# B&R Automation Studio project mappFramework (part 4)

#### FileMgr.st
```iecst
//***********************************************************************
// Copyright: B&R Industrial Automation GmbH
// Author: B&R Industrial Automation GmbH
// Created: April 12, 2022
// Description: Task for file management
//***********************************************************************

PROGRAM _INIT

	// Inititialize mapp function block
	MpFileManagerUIConnect.DeviceList.DeviceNames[0] := 'USER';
	MpFileManagerUIConnect.DeviceList.DeviceNames[1] := 'mappRecipeFiles';
	MpFileManagerUIConnect.DeviceList.DeviceNames[2] := 'mappAuditFiles';
	MpFileManagerUIConnect.DeviceList.DeviceNames[3] := 'mappReportFiles';
	MpFileManagerUIConnect.DeviceList.DeviceNames[4] := 'mappBackupFiles';
	MpFileManagerUIConnect.DeviceList.DeviceNames[5] := 'mappAlarmXFiles';
	MpFileManagerUIConnect.DeviceList.DeviceNames[6] := 'mappUserXFiles';
	MpFileManagerUISys.Enable := TRUE;
	MpFileManagerUISys.MpLink := ADR(gMpLinkFileManagerUIFile);
	MpFileManagerUISys.UIConnect := ADR(MpFileManagerUIConnect);
	MpFileManagerUISys.UISetup.FileListSize := SIZEOF(MpFileManagerUIConnect.File.List.Items) / SIZEOF(MpFileManagerUIConnect.File.List.Items[0]);
	MpFileManagerUISys();

	HmiFile.Status.DeleteStep := FILE_DISABLED;

	// Restored the retained values to the FIFO settings
	HmiFile.Parameters.Fifo := FifoSettingsRetain;
	// If the FIFO is disabled and parameters are 0, set default values
	IF NOT HmiFile.Parameters.Fifo.Enable THEN
		IF HmiFile.Parameters.Fifo.MaxFolderSize = 0 THEN
			HmiFile.Parameters.Fifo.MaxFolderSize := 1000;
		END_IF
		IF HmiFile.Parameters.Fifo.MaxNumberOfFiles = 0 THEN
			HmiFile.Parameters.Fifo.MaxNumberOfFiles := 20;
		END_IF
		IF HmiFile.Parameters.Fifo.ScanInterval = 0 THEN
			HmiFile.Parameters.Fifo.ScanInterval := 60;
		END_IF
		IF HmiFile.Parameters.Fifo.DeviceName = '' THEN
			HmiFile.Parameters.Fifo.DeviceName := 'USER';
		END_IF
	END_IF

	// Initialize which folders should exist
	PathCheck.DeviceList := MpFileManagerUIConnect.DeviceList;

	PathCheck.PrgName[0] := 'RecipeMgr';
	PathCheck.PrgName[1] := 'AuditMgr';
	PathCheck.PrgName[2] := 'ReportMgr';
	PathCheck.PrgName[3] := 'BackupMgr';
	PathCheck.PrgName[4] := 'AlarmMgr';
	PathCheck.PrgName[5] := 'UserXMgr';
	PathCheck.PrgName[6] := 'UsbMgr';
	PathCheck.PrgName[7] := 'UsbMgr';

	PathCheck.Folder[0] := 'Recipe';
	PathCheck.Folder[1] := 'Audit';
	PathCheck.Folder[2] := 'Report';
	PathCheck.Folder[3] := 'Backup';
	PathCheck.Folder[4] := 'AlarmX';
	PathCheck.Folder[5] := 'UserX';

	HmiFile.Status.DeviceDataProvider[0] := '{"value":"USER","text":"UserPath"}';
	HmiFile.Status.DeviceDataProvider[1] := '{"value":"mappRecipeFiles","text":"mappRecipeFiles"}';
	HmiFile.Status.DeviceDataProvider[2] := '{"value":"mappAuditFiles","text":"mappAuditFiles"}';
	HmiFile.Status.DeviceDataProvider[3] := '{"value":"mappReportFiles","text":"mappReportFiles"}';
	HmiFile.Status.DeviceDataProvider[4] := '{"value":"mappBackupFiles","text":"mappBackupFiles"}';
	HmiFile.Status.DeviceDataProvider[5] := '{"value":"mappAlarmXFiles","text":"mappAlarmXFiles"}';
	HmiFile.Status.DeviceDataProvider[6] := '{"value":"mappUserXFiles","text":"mappUserXFiles"}';

	// Calculate offset for potential additional USB devices
	FOR i := 0 TO ((SIZEOF(MpFileManagerUIConnect.DeviceList.DeviceNames) / SIZEOF(MpFileManagerUIConnect.DeviceList.DeviceNames[0])) - 1) DO
		IF MpFileManagerUIConnect.DeviceList.DeviceNames[i] <> '' THEN
			USBOffset := USBOffset + 1;
		END_IF
	END_FOR

END_PROGRAM

PROGRAM _CYCLIC

	// Call all cyclic actions
	FormatDeviceDataProvider;
	FileManager;
	FIFOOperation;

	// Error reset
	IF NOT MpFileManagerUISys.Error THEN
		MpFileManagerUISys.ErrorReset := FALSE;
	END_IF

	// Assign MpLinks and address references
	MpFileManagerUISys.MpLink := ADR(gMpLinkFileManagerUIFile);
	MpFileManagerUISys.UIConnect := ADR(MpFileManagerUIConnect);
	MpFileManagerUI_FIFO.MpLink := ADR(gMpLinkFileManagerUIFile_FIFO);

	// Call function blocks
	MpFileManagerUISys();
	MpFileManagerUI_FIFO();

END_PROGRAM

PROGRAM _EXIT

	// Disable the function blocks to unlink the MpLink
	MpFileManagerUISys.Enable := FALSE;
	MpFileManagerUI_FIFO.Enable := FALSE;

	// Call function blocks
	MpFileManagerUISys();
	MpFileManagerUI_FIFO();

END_PROGRAM
```

#### HMIActions.st
```iecst
ACTION FormatDeviceDataProvider:

	// Select CF device if USB device is not available
	FOR i := 0 TO IDX_USB_DEV_LIST DO
		tempIdx := (i + USBOffset);

		IF gUSBAvailable[i] THEN

			HmiFile.Status.DeviceDataProvider[tempIdx] := '{"value":"USB';
			brsitoa(i + 1, ADR(HmiFile.Status.DeviceDataProvider[tempIdx]) + brsstrlen(ADR(HmiFile.Status.DeviceDataProvider[tempIdx])));

			brsstrcat(ADR(HmiFile.Status.DeviceDataProvider[tempIdx]), ADR('","text":"USB'));
			brsitoa(i + 1, ADR(HmiFile.Status.DeviceDataProvider[tempIdx]) + brsstrlen(ADR(HmiFile.Status.DeviceDataProvider[tempIdx])));
			brsstrcat(ADR(HmiFile.Status.DeviceDataProvider[tempIdx]), ADR('"}'));

			PathCheck.DeviceList.DeviceNames[tempIdx] := 'USB';
			brsitoa(i + 1, ADR(PathCheck.DeviceList.DeviceNames[tempIdx]) + brsstrlen(ADR(PathCheck.DeviceList.DeviceNames[tempIdx])));
		ELSE
			brsmemset(ADR(HmiFile.Status.DeviceDataProvider[tempIdx]), 0, SIZEOF(HmiFile.Status.DeviceDataProvider[tempIdx]));
			brsmemset(ADR(PathCheck.DeviceList.DeviceNames[tempIdx]), 0, SIZEOF(PathCheck.DeviceList.DeviceNames[tempIdx]));
		END_IF
	END_FOR

	//Check initilized folder for existance and remove any from the device list that don't exist
	MaxDeviceNameIndex := ((SIZEOF(MpFileManagerUIConnect.DeviceList.DeviceNames) / SIZEOF(MpFileManagerUIConnect.DeviceList.DeviceNames[0])) - 1);
	NextOpenIndex := 0;
	FOR index := 0 TO MaxDeviceNameIndex DO
		IdentStatus := ST_ident(ADR(PathCheck.PrgName[index]),0,ADR(Ident));
		//Assign device name to next available slot in table according to if the path is valid
		IF (IdentStatus = 0) THEN		//path is valid
			MpFileManagerUIConnect.DeviceList.DeviceNames[NextOpenIndex] := PathCheck.DeviceList.DeviceNames[index + 1];
			NextOpenIndex := NextOpenIndex + 1;
		END_IF;
		//Clear the remaining index slots with invalid path checks
		IF index > NextOpenIndex THEN
			MpFileManagerUIConnect.DeviceList.DeviceNames[index] := '';
		END_IF
	END_FOR;

	// Configure visible device list
	HmiFile.Status.TableConfig[0] := '{ "specRows": [{"from":';
	FOR i := 0 TO MaxDeviceNameIndex DO
		IF MpFileManagerUIConnect.DeviceList.DeviceNames[i] <> '' THEN
			DeviceCount := i + 1;
		END_IF
	END_FOR
	brsitoa((DeviceCount), ADR(HmiFile.Status.TableConfig[0]) + brsstrlen(ADR(HmiFile.Status.TableConfig[0])));
	brsstrcat(ADR(HmiFile.Status.TableConfig[0]), ADR(',"to":9, "visible":false}]}'));

	// Configure visible file list
	HmiFile.Status.TableConfig[1] := '{ "specRows": [{"from":';
	brsitoa((MpFileManagerUIConnect.File.PathInfo.FileCount + MpFileManagerUIConnect.File.PathInfo.FolderCount), ADR(HmiFile.Status.TableConfig[1]) + brsstrlen(ADR(HmiFile.Status.TableConfig[1])));
	brsstrcat(ADR(HmiFile.Status.TableConfig[1]), ADR(',"to":49, "visible":false}]}'));

	// Create device data provider for FIFO drop down
	FOR i := 0 TO MaxDeviceNameIndex DO
		IF (MpFileManagerUIConnect.DeviceList.DeviceNames[i] <> '') THEN
			HmiFile.Status.DeviceDataProvider[i] := '{"value":"';
			brsstrcat(ADR(HmiFile.Status.DeviceDataProvider[i]), ADR(MpFileManagerUIConnect.DeviceList.DeviceNames[i]));
			brsstrcat(ADR(HmiFile.Status.DeviceDataProvider[i]), ADR('","text":"'));
			brsstrcat(ADR(HmiFile.Status.DeviceDataProvider[i]), ADR(MpFileManagerUIConnect.DeviceList.DeviceNames[i]));
			brsstrcat(ADR(HmiFile.Status.DeviceDataProvider[i]), ADR('"}'));
		ELSE
			brsmemset(ADR(HmiFile.Status.DeviceDataProvider[i]), 0, SIZEOF(HmiFile.Status.DeviceDataProvider[i]));
		END_IF
	END_FOR

END_ACTION

ACTION FileManager:

	MpFileManagerUI_0.MpLink := ADR(gMpLinkFileManagerUIFile);
	MpFileManagerUI_0.UIConnect := ADR(MpFileManagerUIConnect);
	MpFileManagerUI_0();

	FOR i := 0 TO ((SIZEOF(HmiFile.Status.FileNames)/SIZEOF(HmiFile.Status.FileNames[0])) - 1) DO
		HmiFile.Status.FileNames[i] := MpFileManagerUIConnect.File.List.Items[i].Name;
		HmiFile.Status.TimeStamps[i] := MpFileManagerUIConnect.File.List.Items[i].LastModified;
		HmiFile.Status.Size[i] := REAL_TO_UDINT(UDINT_TO_REAL(MpFileManagerUIConnect.File.List.Items[i].Size) * 0.001);

		// Set image array based on item type
		IF MpFileManagerUIConnect.File.List.Items[i].IsFolder THEN
			HmiFile.Status.Type[i] := FOLDER;
		ELSIF NOT MpFileManagerUIConnect.File.List.Items[i].IsFolder AND MpFileManagerUIConnect.File.List.Items[i].IsSelected THEN
			HmiFile.Status.Type[i] := FILE_SELECTED;
		ELSE
			HmiFile.Status.Type[i] := FILE;
		END_IF

		// Set file selected when the table is clicked Single and MultiSelect
		IF (MpFileManagerUIConnect.File.MultiSelect = FALSE) THEN
			MpFileManagerUIConnect.File.List.Items[i].IsSelected := (i = HmiFile.Status.SelectedIndex);
		ELSIF (MpFileManagerUIConnect.File.MultiSelect = TRUE) AND (HmiFile.Commands.MultiSelect = TRUE) THEN
			IF (i = HmiFile.Status.SelectedIndex) AND NOT MpFileManagerUIConnect.File.List.Items[i].IsSelected THEN
				MpFileManagerUIConnect.File.List.Items[i].IsSelected := TRUE;
				HmiFile.Commands.MultiSelect := FALSE;
			ELSIF (i = HmiFile.Status.SelectedIndex) AND MpFileManagerUIConnect.File.List.Items[i].IsSelected THEN
				MpFileManagerUIConnect.File.List.Items[i].IsSelected := FALSE;
				HmiFile.Commands.MultiSelect := FALSE;
			END_IF
		END_IF
	END_FOR

	// Read currently selected device name for HMI
	IF (MpFileManagerUIConnect.DeviceList.SelectedIndex >= (SIZEOF(MpFileManagerUIConnect.DeviceList.DeviceNames) / SIZEOF(MpFileManagerUIConnect.DeviceList.DeviceNames[0]))) THEN
		MpFileManagerUIConnect.DeviceList.SelectedIndex := 0;
	END_IF
	HmiFile.Status.DeviceName := MpFileManagerUIConnect.DeviceList.DeviceNames[MpFileManagerUIConnect.DeviceList.SelectedIndex];

	// Read if current selected object is folder
	IF (HmiFile.Status.SelectedIndex >= (SIZEOF(MpFileManagerUIConnect.File.List.Items) / SIZEOF(MpFileManagerUIConnect.File.List.Items[0]))) THEN
		HmiFile.Status.SelectedIndex := 0;
	END_IF
	HmiFile.Status.IsFolder := MpFileManagerUIConnect.File.List.Items[HmiFile.Status.SelectedIndex].IsFolder;

	// Control the folder structure when entering and leaving folders
	IF (HmiFile.Commands.EnterFolder) AND MpFileManagerUIConnect.File.List.Items[HmiFile.Status.SelectedIndex].IsFolder THEN
		HmiFile.Commands.EnterFolder := FALSE;
		MpFileManagerUIConnect.File.EnterFolder := TRUE;
		FolderDepthCount := FolderDepthCount + 1;
	ELSE
		HmiFile.Commands.EnterFolder := FALSE;
	END_IF

	IF EDGEPOS(HmiFile.Commands.FolderUp) AND (HmiFile.Status.BackButton > 0) THEN
		HmiFile.Commands.FolderUp := FALSE;
		MpFileManagerUIConnect.File.FolderUp := TRUE;
		FolderDepthCount := FolderDepthCount - 1;
	END_IF

	HmiFile.Status.BackButton := (FolderDepthCount > 0);
	HmiFile.Status.DefaultFileSelected := ((MpFileManagerUIConnect.File.List.Items[HmiFile.Status.SelectedIndex].Name = CONCAT(DEFAULT_PARAMETERS,PARAMETERS_FILE_EXTENSION)) OR
																				(MpFileManagerUIConnect.File.List.Items[HmiFile.Status.SelectedIndex].Name = CONCAT(DEFAULT_MACHINE_CONFIGURATION,
																				MACHINE_CONFIG_FILE_EXTENSION))) AND MpFileManagerUIConnect.DeviceList.SelectedIndex = 0;

END_ACTION
```

### Package Logical/Infrastructure/Usb - Package for USB handling for mapp Framework

### Program Logical/Infrastructure/Usb/UsbMgr (IEC)

#### UsbMgr.st - Cyclic code
```iecst
//*********************************************************************************
// Copyright: B&R Industrial Automation GmbH
// Author: B&R Industrial Automation GmbH
// Created: April 12, 2022
// Description: This task automatically detects and (un)links USB storage devices
//*********************************************************************************

PROGRAM _INIT
END_PROGRAM

PROGRAM _CYCLIC

	CASE StateMachine OF
		// -----------------------------------------------------------------------------------------------------------
		// Wait state
		// -----------------------------------------------------------------------------------------------------------
		USB_WAIT:
			// Refresh USB data every X seconds when enabled
			Node := 1;
			USB.Status := ERR_OK;
			IF USB.Cmd.AutoScan THEN
				RefreshTimer(IN := 1, PT := USB.Par.RefreshInterval);
				// Get new USB data
				IF(RefreshTimer.Q) THEN
					RefreshTimer(IN := 0);
					USB.Status := ERR_FUB_BUSY;
					brsmemset(ADR(UsbData), 0, SIZEOF(UsbData));
					StateMachine := USB_CREATE_NODE_ID_LIST;
				END_IF
			ELSE
				RefreshTimer(IN := 0);
			END_IF
			// Refresh USB data every X seconds when enabled
			IF USB.Cmd.ErrorReset THEN
				StateMachine := USB_ERROR;
			END_IF

			FOR i := 0 TO IDX_USB_DEV_LIST DO
				gUSBAvailable[i] := USB.Par.IsConnected[i+1];
			END_FOR

			// -----------------------------------------------------------------------------------------------------------
			// Get USB device list
			// -----------------------------------------------------------------------------------------------------------
		USB_CREATE_NODE_ID_LIST:
			GetUsbNodeList.enable := 1;
			GetUsbNodeList.pBuffer := ADR(NodeIdBuffer);
			GetUsbNodeList.bufferSize := SIZEOF(NodeIdBuffer);
			GetUsbNodeList.filterInterfaceClass := asusb_CLASS_MASS_STORAGE;
			GetUsbNodeList.filterInterfaceSubClass := 0;
			GetUsbNodeList;

			// --------------------------------------------------------------------------------------------------------------------
			// Success
			IF GetUsbNodeList.status = 0 THEN
				StateMachine := USB_READ_DEVICE_DATA;
				Node := 1;
				// No USB devices found
			ELSIF GetUsbNodeList.status = asusbERR_USB_NOTFOUND THEN
				// Unlink old device if it is gone now otherwise wait for next round
				FOR i:=1 TO MAX_IDX_USB_DEV_LIST DO
					IF(USB.Par.IsConnected[i]) THEN
						Node := 1;
						StateMachine := USB_CHECK_LINKED;
						RETURN;
					END_IF
				END_FOR;
				StateMachine := USB_WAIT;
				// Error
			ELSIF GetUsbNodeList.status <> ERR_FUB_BUSY THEN
				USB.Status := GetUsbNodeList.status;
				USB.Err.State := StateMachine;
				IF GetUsbNodeList.status = asusbERR_BUFSIZE THEN
					USB.Err.Text := 'maximum number of devices reached';
				ELSE
					USB.Err.Text := 'error getting device list';
				END_IF;
				StateMachine := USB_ERROR;
			END_IF;
			// -----------------------------------------------------------------------------------------------------------
			// Get device information
			// -----------------------------------------------------------------------------------------------------------
		USB_READ_DEVICE_DATA:
			GetUsbNode.enable := 1;
			GetUsbNode.nodeId := NodeIdBuffer[Node];
			GetUsbNode.pBuffer := ADR(UsbData[Node]);
			GetUsbNode.bufferSize := SIZEOF (UsbData[Node]);
			GetUsbNode;

			// --------------------------------------------------------------------------------------------------------------------
			// Success
			IF GetUsbNode.status = 0 THEN
				// Make sure we have enough space to store USB data, proceed with next StateMachine when all devices are detetced
				IF (Node = GetUsbNodeList.listNodes) OR (Node = MAX_IDX_USB_DEV_LIST) THEN
					Node := 1;
					StateMachine := USB_CHECK_LINKED;
					// Get next USB device
				ELSE
					Node := Node + 1;
				END_IF;
				// Error
			ELSIF GetUsbNode.status <> ERR_FUB_BUSY THEN
				USB.Status := GetUsbNode.status;
				USB.Err.State := StateMachine;
				USB.Err.Text := 'error getting device data';
				StateMachine := USB_ERROR;
			END_IF;
			// -----------------------------------------------------------------------------------------------------------
			// Check if linked device are still present
			// -----------------------------------------------------------------------------------------------------------
		USB_CHECK_LINKED:
			// Proceed to new devices when last device was checked
			IF(Node > MAX_IDX_USB_DEV_LIST) THEN
				Node := 1;
				StateMachine := USB_LINK_NEW;
				RETURN;
			END_IF

			// -----------------------------------------------------------------------------------------------------------
			// Check if device is still active
			IsLinked := FALSE;
			FOR i:=1 TO MAX_IDX_USB_DEV_LIST DO
				// Compare old and new data
				IF(brsmemcmp(ADR(UsbDataOld[Node]), ADR(UsbData[i]), SIZEOF(UsbData[i])) = 0) AND
					(NOT USB.Par.IgnoreDongle OR (USB.Par.IgnoreDongle AND UsbData[i].productId <> BrProductId AND UsbData[i].vendorId <> BrVendorId)) THEN
					// Clear data, mark as linked and EXIT loop
					brsmemset(ADR(UsbData[i]), 0, SIZEOF(UsbData[i]));
					IsLinked := TRUE;
					EXIT;
				END_IF
			END_FOR;

			// -----------------------------------------------------------------------------------------------------------
			// Find next linked device
			IF(IsLinked OR UsbDataOld[Node].interfaceClass = 0) THEN
				IF(Node < MAX_IDX_USB_DEV_LIST) THEN
					Node := Node + 1;
					WHILE(Node < MAX_IDX_USB_DEV_LIST AND UsbDataOld[Node].interfaceClass = 0) DO
						Node := Node + 1;
					END_WHILE;
					IF(Node = MAX_IDX_USB_DEV_LIST AND UsbDataOld[Node].interfaceClass = 0) THEN
						Node := Node + 1;
					END_IF
				ELSE
					Node := Node + 1;
				END_IF
				// Unlink device if it is missing
			ELSE
				StateMachine := USB_UNLINK_DEVICE;
			END_IF
			// -----------------------------------------------------------------------------------------------------------
			// Link new devices
			// -----------------------------------------------------------------------------------------------------------
		USB_LINK_NEW:
			// Return to wait state when last device was checked
			IF(Node > MAX_IDX_USB_DEV_LIST) THEN
				StateMachine := USB_WAIT;
				RETURN;
			END_IF

			// -----------------------------------------------------------------------------------------------------------
			// Find next new device
			IF(UsbData[Node].interfaceClass <> 0) THEN
				IF(USB.Par.IgnoreDongle OR (UsbData[Node].productId <> BrProductId AND UsbData[Node].vendorId <> BrVendorId)) THEN
					StateMachine := USB_LINK_DEVICE;
					RETURN;
				END_IF
			END_IF
			Node := Node + 1;
			// -----------------------------------------------------------------------------------------------------------
			// Link device
			// -----------------------------------------------------------------------------------------------------------
		USB_LINK_DEVICE:
			// Find empty slot
			FOR i:=1 TO MAX_IDX_USB_DEV_LIST DO
				IF(UsbDataOld[i].interfaceClass = 0) THEN
					EXIT;
				END_IF
			END_FOR;
			// No more slot available
			IF(i = MAX_IDX_USB_DEV_LIST AND UsbDataOld[i].interfaceClass <> 0) THEN
				USB.Status := ERR_MAX_DEVICE;
				USB.Err.State := StateMachine;
				USB.Err.Text := 'maximum number of device reached';
				StateMachine := USB_ERROR;
				RETURN;
			END_IF
			// Create device string
			brsstrcpy(ADR(DevicePara), ADR('/DEVICE='));
			brsstrcat(ADR(DevicePara), ADR(UsbData[Node].ifName));
			brsstrcpy(ADR(DeviceName), ADR('USB'));
			brsitoa(i, ADR(tmpSTR));
			brsstrcat(ADR(DeviceName), ADR(tmpSTR));
			// Link device
			DevLinkSys.enable := 1;
			DevLinkSys.pDevice := ADR(DeviceName);
			DevLinkSys.pParam := ADR(DevicePara);
			DevLinkSys;

			// --------------------------------------------------------------------------------------------------------------------
			// Success
			IF DevLinkSys.status = 0 THEN
				// Store data for new device
				brsmemcpy(ADR(UsbDataOld[i]), ADR(UsbData[Node]), SIZEOF(UsbData[Node]));
				USB.Par.IsConnected[i] := TRUE;
				LinkHandle[i] := DevLinkSys.handle;
				Node := Node + 1;
				StateMachine := USB_LINK_NEW;
				// Error
			ELSIF DevLinkSys.status <> ERR_FUB_BUSY THEN
				USB.Status := DevLinkSys.status;
				USB.Err.State := StateMachine;
				USB.Err.Text := 'error linking device';
				StateMachine := USB_ERROR;
			END_IF;
			// -----------------------------------------------------------------------------------------------------------
			// UnLink device
			// -----------------------------------------------------------------------------------------------------------
		USB_UNLINK_DEVICE:
			DevUnlinkSys.enable := 1;
			DevUnlinkSys.handle := LinkHandle[Node];
			DevUnlinkSys;

			// --------------------------------------------------------------------------------------------------------------------
			// Success
			IF DevUnlinkSys.status = 0 THEN
				// Clear data
				brsmemset(ADR(UsbDataOld[Node]), 0, SIZEOF(UsbDataOld[Node]));
				USB.Par.IsConnected[Node] := FALSE;
				LinkHandle[Node] := 0;
				// Find next linked device
				WHILE(Node < MAX_IDX_USB_DEV_LIST AND UsbDataOld[Node].interfaceClass = 0) DO
					Node := Node + 1;
				END_WHILE;
				IF(Node = MAX_IDX_USB_DEV_LIST AND UsbDataOld[Node].interfaceClass = 0) THEN
					Node := Node + 1;
				END_IF
				StateMachine := USB_CHECK_LINKED;
				// Error
			ELSIF DevUnlinkSys.status <> ERR_FUB_BUSY THEN
				// Clear data
				brsmemset(ADR(UsbDataOld[Node]), 0, SIZEOF(UsbDataOld[Node]));
				USB.Par.IsConnected[Node] := FALSE;
				LinkHandle[Node] := 0;

				brsitoa(Node, ADR(tmpSTR));
				USB.Status := DevUnlinkSys.status;
				USB.Err.State := StateMachine;
				USB.Err.Text := 'error unlinking device no ';
				brsstrcat(ADR(USB.Err.Text), ADR(tmpSTR));
				StateMachine := USB_ERROR;
			END_IF;
			// -----------------------------------------------------------------------------------------------------------
			// Error state
			// -----------------------------------------------------------------------------------------------------------
		USB_ERROR:
			// Get more error information
			IF(USB.Status = 0) THEN
				USB.Status := FileIoGetSysError();
			END_IF

			// Unlink device
			IF(USB.Err.State = USB_LINK_DEVICE) THEN
				DevUnlinkSys.enable := 1;
				DevUnlinkSys.handle := DevLinkSys.handle;
				DevUnlinkSys;
			END_IF

			// Reset error
			IF(USB.Cmd.ErrorReset AND DevUnlinkSys.status <> ERR_FUB_BUSY) THEN
				USB.Cmd.ErrorReset := FALSE;
				brsmemset(ADR(USB.Err), 0, SIZEOF(USB.Err));
				StateMachine := USB_WAIT;
			END_IF
	END_CASE;

END_PROGRAM

PROGRAM _EXIT
	FOR i:=1 TO MAX_IDX_USB_DEV_LIST DO
		REPEAT
			DevUnlinkSys.enable := 1;
			DevUnlinkSys.handle := LinkHandle[i];
			DevUnlinkSys;
			UNTIL DevUnlinkSys.status <> ERR_FUB_BUSY
		END_REPEAT;
	END_FOR;
END_PROGRAM
```

#### UsbMgr.typ
```iecst
TYPE
	UsbStateEnum :
		(
		USB_WAIT, (*Wait for starting the Function chain*)
		USB_CREATE_NODE_ID_LIST, (*Create a list of Node-IDs from all active USB devices*)
		USB_READ_DEVICE_DATA, (*Read out the specific data from the Node-IDs*)
		USB_CHECK_LINKED, (*Check if device is still connected*)
		USB_LINK_NEW,
		USB_LINK_DEVICE, (*Link file device*)
		USB_UNLINK_DEVICE, (*Unlink the File Device from specific path*)
		USB_ERROR (*Jump to this step in every case of Error occuring in the Function chain*)
		);
	UsbCmdType : 	STRUCT
		AutoScan : BOOL := TRUE; (*Scan USB ports automatically*)
		ErrorReset : BOOL; (*Reset error*)
	END_STRUCT;
	UsbParType : 	STRUCT
		IgnoreDongle : BOOL := TRUE; (*Ignoe B&R license dongle*)
		RefreshInterval : UINT := 300; (*Intervall timer for USB device refresh*)
		IsConnected : ARRAY[0..MAX_IDX_USB_DEV_LIST]OF BOOL; (*Shows if a USB stick is connected*)
	END_STRUCT;
	UsbErrType : 	STRUCT
		State : UsbStateEnum; (*State where the error occured*)
		Text : STRING[80]; (*Error text*)
	END_STRUCT;
	UsbMainType : 	STRUCT
		Cmd : UsbCmdType; (*Command structure*)
		Par : UsbParType; (*Parameter structure*)
		Err : UsbErrType; (*Error structure*)
		Status : UINT; (*Current status*)
	END_STRUCT;
END_TYPE
```

#### UsbMgr.var - Data for read_data Task
```iecst
(*Function Blocks*)
VAR
	RefreshTimer : TON;
	GetUsbNodeList : UsbNodeListGet; (*Type of FUB UsbNodeListGet*)
	GetUsbNode : UsbNodeGet; (*Type of FUB UsbNodeGet*)
	DevLinkSys : DevLink; (*Type of FUB DevLink*)
	DevUnlinkSys : DevUnlink; (*Type of FUB DevUnlink*)
END_VAR
(*Constants*)
VAR CONSTANT
	BrVendorId : UINT := 1615; (*B&R vendor id*)
	BrProductId : UINT := 1001; (*B&R dongle product id*)
	ERR_MAX_DEVICE : UINT := 50000; (*Maximum number of dongles reached*)
END_VAR
(*Structure Types*)
VAR
	USB : UsbMainType;
	StateMachine : UsbStateEnum; (*State machine*)
	UsbData : ARRAY[1..MAX_IDX_USB_DEV_LIST] OF usbNode_typ; (*Data of all available USB devices*)
	UsbDataOld : ARRAY[1..MAX_IDX_USB_DEV_LIST] OF usbNode_typ; (*Old data of all available USB devices*)
END_VAR
(*Variables*)
VAR
	DevicePara : STRING[80]; (*Connection path of USB device*)
	DeviceName : STRING[40]; (*Connection path of USB device*)
	LinkHandle : ARRAY[1..MAX_IDX_USB_DEV_LIST] OF UDINT; (*Link handle for USB device*)
	NodeIdBuffer : ARRAY[1..MAX_IDX_USB_DEV_LIST] OF UDINT; (*Different nodeIDs saved in array-elements*)
	IsLinked : BOOL; (*Helper variable that indicates that a USB stick is linked*)
	Node : USINT; (*Node number*)
	i : USINT;
	tmpSTR : STRING[10];
END_VAR
```

### Package Logical/Infrastructure/Recipe - Package for mapp Recipe Framework

### Program Logical/Infrastructure/Recipe/RecipeMgr (IEC) - Recipe manager

#### RecipeMgr.typ
```iecst
(*Structure types*)

TYPE
	RecipeHmiInterfaceType : 	STRUCT  (*Structure to hold commands, parameters and status from the HMI*)
		Commands : RecipeCommandsType; (*Structure to hold the commands from the HMI*)
		Parameters : RecipeParametersType; (*Structure to hold the parameters for the HMI*)
		Status : RecipeStatusType; (*Structure to hold status information from the mapp View HMI*)
	END_STRUCT;
	RecipeCommandsType : 	STRUCT  (*Structure to hold the commands from the HMI*)
		LoadRecipe : BOOL; (*Load recipe*)
		SaveSelectedRecipe : BOOL; (*Save the selected recipe (which is not necessarily the active recipe)*)
		CreateRecipe : BOOL; (*Create recipe*)
		ResetPreview : BOOL; (*Reset the preview to empty/zeros in the event of an invalid recipe*)
	END_STRUCT;
	RecipeParametersType : 	STRUCT  (*Structure to hold the parameters for the HMI*)
		Category : STRING[30]; (*Current category*)
		DeviceName : STRING[50]; (*Selected file device name*)
		FileName : STRING[255]; (*Recipe file name*)
	END_STRUCT;
	RecipeStatusType : 	STRUCT  (*Structure to hold status information from the mapp View HMI*)
		PreviewCase : PreviewCaseEnum; (*State machine step for loading previews*)
		HMIcommand : RecipeHmiStepEnum; (*State machine step for HMI commands*)
		LastLoadedConfigRecipe : STRING[255]; (*Last loaded configuration recipe*)
		LastLoadedProductRecipe : STRING[255]; (*Last loaded product recipe*)
		ProductRecipeLoaded : BOOL; (*Product recipe was loaded*)
		ConfigRecipeLoaded : BOOL; (*Config recipe was loaded*)
		PreviousRangeStart : REAL; (*Scroll range temp variables*)
		PreviousRangeEnd : REAL; (*Scroll range temp variables*)
		LastMaxSelection : UINT; (*The previous maximum number of recipes*)
		SelectedIndex : UINT; (*The currently selected index*)
		LastSelectedIndex : UINT; (*The previous selected index*)
		LastStatus : MpRecipeUIStatusEnum; (*The previous UI status*)
		EditDialogOpened : BOOL; (*Flag that the edit dialog box was opened*)
		CreateDialogOpened : BOOL; (*Flag that the create dialog box was opened*)
		DefaultConfig : STRING[255]; (*Name of the default configuration*)
		DefaultRecipe : STRING[255]; (*Name of the default recipe*)
		FileDuplicate : BOOL; (*Recipe file already exists, warn the user.*)
		FilesAvailable : BOOL; (*Control access to widget when no files are available*)
		InvalidRecipe : BOOL; (*The selected recipe cannot be previewed*)
		LoadingRecipeList : BOOL; (*The recipe list is loading*)
		MachineSettingsRecipeMissing : BOOL; (*Flag for if the default machine settings recipe is not present*)
		ParameterRecipeMissing : BOOL; (*Flag for if the default parameters recipe is not present*)
		DeviceValid : BOOL; (*Flag for whether FileDevice is valid. Prevents user from being prompted to load default recipe.*)
		LoadAllowed : BOOL; (*Flag for whether you can load a recipe. Recipe must exist and be valid. *)
		DeviceDataProvider : ARRAY[0..MAX_IDX_FILE_DEV]OF STRING[100]; (*File device data provider*)
		TableConfig : STRING[120]; (*Table configuration *)
		SelectedRecipe : STRING[255]; (*The name of the selected recipe*)
		DefaultRecipeSelected : BOOL; (*The default recipe is selected*)
		RecipeContentLoaded : BOOL; (*Recipe content is loading and previous selection is restored*)
	END_STRUCT;
	RecipeRetainType : 	STRUCT  (*Structure to hold parameters for retain after restart *)
		LastLoadedConfigRecipe : STRING[255]; (*Last loaded configuration recipe*)
		LastLoadedProductRecipe : STRING[255]; (*Last loaded product recipe*)
	END_STRUCT;
	ParametersType : 	STRUCT  (*Demo / starter structure for machine parameters*)
		AddParametersHere1 : BOOL; (*Add your parameteres here *)
		AddParametersHere2 : STRING[80]; (*Add your parameteres here *)
		AddParametersHere3 : REAL; (*Add your parameteres here *)
		AddParametersHere4 : REAL; (*Add your parameteres here *)
		AddParametersHere5 : REAL; (*Add your parameteres here *)
	END_STRUCT;
	MachineSettingsType : 	STRUCT  (*Demo / starter structure for machine configuration settings*)
		AddMachineSettingsHere1 : USINT; (*Add your settings here*)
		AddMachineSettingsHere2 : DINT; (*Add your settings here*)
		AddMachineSettingsHere3 : BOOL; (*Add your settings here*)
		AddMachineSettingsHere4 : REAL; (*Add your settings here*)
		AddMachineSettingsHere5 : UINT; (*Add your settings here*)
	END_STRUCT;
END_TYPE

(*Enumerations*)

TYPE
	RecipeHmiStepEnum :
		( (*State machine step for HMI commands*)
		REC_HMI_WAIT, (*Wait*)
		REC_HMI_LOAD, (*Load recipe*)
		REC_HMI_SAVE, (*Save recipe*)
		REC_HMI_CREATE, (*Create recipe*)
		REC_HMI_RESET_PREVIEW (*Reset the preview values to 0 / empty*)
		);
	PreviewCaseEnum :
		( (*State machine step for loading Preview*)
		PREVIEW_WAIT, (*Wait*)
		PREVIEW_LOAD, (*Load recipe*)
		PREVIEW_CHANGE (*Show new preview*)
		);
END_TYPE
```

#### RecipeMgr.var
```iecst
(*Function Blocks*)
VAR
	MpRecipeSys : MpRecipeXml; (*MpRecipe instance*)
	MpRecipeRegPar_PreviewPar : MpRecipeRegPar; (*MpRecipeRegPar instance for ParametersPreview variable*)
	MpRecipeRegPar_PreviewCfg : MpRecipeRegPar; (*MpRecipeRegPar instance for MachineSettingsPreview*)
	MpRecipeUISys : MpRecipeUI; (*MpRecupeUI instance*)
	MpFileManagerUIRecipe : MpFileManagerUI; (*MpFileManagerUI instance*)
	DTGetTimeRecipe : DTGetTime; (*DTGetTime instance*)
	DirCreateRecipe : DirCreate; (*DirCreate instance*)
END_VAR
(*Constants*)
VAR CONSTANT
	MAX_IDX_FILE_DEV : USINT := MAX_IDX_USB_DEV_LIST + 1; (*Maximum number of  file devices *)
END_VAR
VAR
	PARAMETERS_RECIPE : STRING[50] := 'Parameters'; (*Value of the DropDownBox selection for the Parameters category*)
	MACHINE_CONFIGURATION_RECIPE : STRING[50] := 'Machine Configuration'; (*Value of the DropDownBox selection for the Machine Configuration category*)
END_VAR
(*Structure Types*)
VAR
	HmiRecipe : RecipeHmiInterfaceType; (*HMI interface structure*)
END_VAR
VAR RETAIN
	HmiRecipeRetain : RecipeRetainType;
END_VAR
VAR
	Parameters : ParametersType; (*Machine parameters. Used by the machine at runtime*)
	ParametersEdit : {REDUND_UNREPLICABLE} ParametersType; (*Machine parameters edit structure. Enables you to edit a recipe that is not currently active*)
	ParametersPreview : ParametersType; (*Machine parameters preview structure. Registered to the recipe. Enables you to preview a recipe that is not currently active.*)
	MachineSettings : MachineSettingsType; (*Machine settings. Used by the machine at runtime.*)
	MachineSettingsEdit : MachineSettingsType; (*Machine settings edit structure. Enables you to edit a recipe that is not currently active*)
	MachineSettingsPreview : MachineSettingsType; (*Machine settings preview structure. Registered to the recipe. Enables you to preview a recipe that is not currently active. *)
	MpRecipeUIConnect : MpRecipeUIConnectType; (*MpRecipeUI connection to the HMI*) (*ParameterFileStep : INT;*)
	MpRecipeUISetup : MpRecipeUISetupType; (*MpRecipeUI setup connection to the HMI*) (*ParameterFileStep : INT;*)
	MpFileManagerUIConnect : MpFileManagerUIConnectType; (*File manager connection to the HMI*)
	Header : MpRecipeXmlHeaderType; (*Header information*)
END_VAR
(*Variables*)
VAR
	i : USINT; (*Index to loop through file devices*)
	temp : STRING[260]; (*Temporary recipe name, used to check for duplicates when creating a new recipe*)
END_VAR
```

#### FileOperations.st
```iecst
ACTION FileCopyOperation:

	// Export/Import recipes to/from USB
    CASE HmiRecipe.Status.CopyStep OF
		REC_COPY_WAIT:
			// Wait for export/import command
            IF (HmiRecipe.Commands.ExportToUSB = TRUE) THEN
                // Check if USB device is available
                IF (brsstrlen(ADR(MpFileManagerUIConnect.DeviceList.DeviceNames[1])) > 0) THEN
					// USB is available proceed with export: select all files on the CF and trigger copy command
                    IF (MpFileManagerUIConnect.DeviceList.SelectedIndex <> 0) THEN
                        MpFileManagerUIConnect.DeviceList.SelectedIndex := 0;
                        MpFileManagerUIConnect.File.MultiSelect := FALSE;
                    ELSIF (MpFileManagerUIConnect.Status = mpFILE_UI_STATUS_IDLE) THEN

                        IF NOT MpFileManagerUIConnect.File.MultiSelect THEN
                            MpFileManagerUIConnect.File.MultiSelect := TRUE;
                            FOR i := 0 TO ((SIZEOF(MpFileManagerUIConnect.File.List.Items) / SIZEOF(MpFileManagerUIConnect.File.List.Items[0])) - 1) DO
                                MpFileManagerUIConnect.File.List.Items[i].IsSelected := TRUE;
                            END_FOR
                        ELSIF (brsstrlen(ADR(MpFileManagerUIConnect.File.List.Items[i].Name)) = 0) THEN
                            // No files to copy, cancel operation
                            HmiRecipe.Commands.ExportToUSB := FALSE;
                        ELSE
                            MpFileManagerUIConnect.File.Copy := TRUE;
							HmiRecipe.Status.CopyStep := REC_COPY_TO_USB;
                            HmiRecipe.Commands.ExportToUSB := FALSE;
                        END_IF

                    END_IF

                ELSE
                    // No USB disk available, cancel operation
                    HmiRecipe.Commands.ExportToUSB := FALSE;
                END_IF

            ELSIF HmiRecipe.Commands.ImportFromUSB THEN
                // Check if USB device is available
                IF (brsstrlen(ADR(MpFileManagerUIConnect.DeviceList.DeviceNames[1])) > 0) THEN
                    // USB is available proceed with import: select all files on the USB and trigger copy command

                    IF (MpFileManagerUIConnect.DeviceList.SelectedIndex <> 1) THEN
                        MpFileManagerUIConnect.DeviceList.SelectedIndex := 1;
                        MpFileManagerUIConnect.File.MultiSelect := FALSE;
                    ELSIF MpFileManagerUIConnect.Status = mpFILE_UI_STATUS_IDLE THEN

                        IF NOT MpFileManagerUIConnect.File.MultiSelect THEN
                            MpFileManagerUIConnect.File.MultiSelect := TRUE;
                            FOR i := 0 TO ((SIZEOF(MpFileManagerUIConnect.File.List.Items)/SIZEOF(MpFileManagerUIConnect.File.List.Items[0])) - 1) DO
                                MpFileManagerUIConnect.File.List.Items[i].IsSelected := TRUE;
                            END_FOR
                        ELSIF (brsstrlen(ADR(MpFileManagerUIConnect.File.List.Items[i].Name)) = 0) THEN
                            // No files to copy, cancel operation
                            HmiRecipe.Commands.ImportFromUSB := FALSE;
                        ELSE
                            MpFileManagerUIConnect.File.Copy := TRUE;
                            HmiRecipe.Status.CopyStep := REC_COPY_FROM_USB;
                            HmiRecipe.Commands.ImportFromUSB := FALSE;
                        END_IF

                    END_IF
                ELSE
                    // No USB disk available, cancel operation
                    HmiRecipe.Commands.ImportFromUSB := FALSE;
                END_IF

            END_IF

		REC_COPY_TO_USB:
			// Navigate to USB device and paste files
            IF (MpFileManagerUIConnect.Status = mpFILE_UI_STATUS_IDLE) THEN

                IF (MpFileManagerUIConnect.DeviceList.SelectedIndex <> 1) THEN
                    MpFileManagerUIConnect.DeviceList.SelectedIndex := 1;
                    MpFileManagerUIConnect.File.MultiSelect := FALSE;
                ELSE
                    MpFileManagerUIConnect.File.Paste := TRUE;
                END_IF

            END_IF

            IF MpFileManagerUIConnect.Status = mpFILE_UI_STATUS_PASTE THEN
                HmiRecipe.Status.CopyStep := REC_COPY_BUSY;
            END_IF

		REC_COPY_FROM_USB:
			// Navigate to CF device and paste files
            IF (MpFileManagerUIConnect.DeviceList.SelectedIndex <> 0) THEN
                MpFileManagerUIConnect.DeviceList.SelectedIndex := 0;
                MpFileManagerUIConnect.File.MultiSelect := FALSE;
            ELSIF (MpFileManagerUIConnect.Status = mpFILE_UI_STATUS_IDLE) THEN
                MpFileManagerUIConnect.File.Paste := TRUE;
            END_IF

            IF (MpFileManagerUIConnect.Status = mpFILE_UI_STATUS_PASTE) THEN
                HmiRecipe.Status.CopyStep := REC_COPY_BUSY;
            END_IF

		REC_COPY_BUSY:
			// Wait for copying done
            IF (MpFileManagerUIConnect.MessageBox.Type = mpFILE_MSG_CONFIRM_OVERWRITE) OR (MpFileManagerUIConnect.MessageBox.Type = mpFILE_MSG_BUSY) THEN
                // TODO: Replace by confirm dialog
                MpFileManagerUIConnect.MessageBox.Confirm := TRUE;
            ELSIF MpFileManagerUIConnect.Status = mpFILE_UI_STATUS_IDLE THEN
                MpRecipeUIConnect.Recipe.Refresh := (MpRecipeUIConnect.Status = mpRECIPE_UI_STATUS_IDLE);
                HmiRecipe.Status.CopyStep := REC_COPY_WAIT;
            END_IF

    END_CASE

END_ACTION
```

#### HMIActions.st
```iecst
ACTION FormatDeviceDataProvider:

	// Select CF device if USB device is not available
	FOR i := 0 TO ((SIZEOF(gUSBAvailable) / SIZEOF(gUSBAvailable[0])) - 1) DO
		IF gUSBAvailable[i] THEN
			HmiRecipe.Status.DeviceDataProvider[i + 1] := '{"value":"USB';
			brsitoa(i + 1, ADR(HmiRecipe.Status.DeviceDataProvider[i + 1]) + brsstrlen(ADR(HmiRecipe.Status.DeviceDataProvider[i + 1])));
			brsstrcat(ADR(HmiRecipe.Status.DeviceDataProvider[i + 1]), ADR('","text":"USB'));
			brsitoa(i + 1, ADR(HmiRecipe.Status.DeviceDataProvider[i + 1]) + brsstrlen(ADR(HmiRecipe.Status.DeviceDataProvider[i + 1])));
			brsstrcat(ADR(HmiRecipe.Status.DeviceDataProvider[i + 1]), ADR('"}'));
			MpFileManagerUIConnect.DeviceList.DeviceNames[i + 1] := 'USB';
			brsitoa(i + 1, ADR(MpFileManagerUIConnect.DeviceList.DeviceNames[i + 1]) + brsstrlen(ADR(MpFileManagerUIConnect.DeviceList.DeviceNames[i + 1])));
		ELSE
			brsmemset(ADR(HmiRecipe.Status.DeviceDataProvider[i + 1]), 0, SIZEOF(HmiRecipe.Status.DeviceDataProvider[i + 1]));
			brsmemset(ADR(MpFileManagerUIConnect.DeviceList.DeviceNames[i + 1]), 0, SIZEOF(MpFileManagerUIConnect.DeviceList.DeviceNames[i + 1]));
		END_IF
	END_FOR

END_ACTION

ACTION LoadStatus:
	// Configure visible recipe list
	IF MpRecipeUIConnect.Recipe.List.Names[0] = '' THEN
		HmiRecipe.Status.TableConfig := '{ "specRows": [{"from":0,"to":19, "visible":false}]}';
	ELSE
		HmiRecipe.Status.TableConfig := '{ "specRows": [{"from":';
		brsitoa(MpRecipeUIConnect.Recipe.List.MaxSelection + 1, ADR(HmiRecipe.Status.TableConfig) + brsstrlen(ADR(HmiRecipe.Status.TableConfig)));
		brsstrcat(ADR(HmiRecipe.Status.TableConfig), ADR(',"to":19, "visible":false}]}'));
	END_IF

	HmiRecipe.Status.FilesAvailable := (MpRecipeUIConnect.Recipe.List.Names[0] <> '');
	HmiRecipe.Status.LoadAllowed := HmiRecipe.Status.FilesAvailable AND NOT HmiRecipe.Status.InvalidRecipe;
	HmiRecipe.Status.DeviceValid := (MpFileManagerUI_0.StatusID <> mpFILE_ERR_INVALID_FILE_DEV);

END_ACTION

ACTION LoadPreview:

	CASE HmiRecipe.Status.PreviewCase OF
		PREVIEW_WAIT:
			// Load preview when a recipe is selected
			IF (MpRecipeUIConnect.Recipe.List.SelectedIndex <> HmiRecipe.Status.LastSelectedIndex) OR (HmiRecipe.Status.LastMaxSelection <> MpRecipeUIConnect.Recipe.List.MaxSelection)
				OR (HmiRecipe.Status.PreviousRangeStart <> MpRecipeUIConnect.Recipe.List.RangeStart) OR (HmiRecipe.Status.PreviousRangeStart <> MpRecipeUIConnect.Recipe.List.RangeStart) THEN
				HmiRecipe.Status.PreviewCase := PREVIEW_LOAD;
			END_IF

		PREVIEW_LOAD:
			// Check selected recipe name is not empty
			IF (brsstrlen(ADR(MpRecipeUIConnect.Recipe.List.Names[MpRecipeUIConnect.Recipe.List.SelectedIndex])) > 0) THEN
				MpRecipe_0.FileName := ADR(MpRecipeUIConnect.Recipe.List.Names[MpRecipeUIConnect.Recipe.List.SelectedIndex]);
				MpRecipe_0.Category := ADR(HmiRecipe.Parameters.Category);
				MpRecipe_0.Load := TRUE;
				HmiRecipe.Status.LastSelectedIndex := MpRecipeUIConnect.Recipe.List.SelectedIndex;
				HmiRecipe.Status.LastMaxSelection := MpRecipeUIConnect.Recipe.List.MaxSelection;
				HmiRecipe.Status.PreviousRangeStart := MpRecipeUIConnect.Recipe.List.RangeStart;
				HmiRecipe.Status.PreviousRangeEnd := MpRecipeUIConnect.Recipe.List.RangeEnd;
				HmiRecipe.Status.InvalidRecipe := FALSE;
				HmiRecipe.Status.PreviewCase := PREVIEW_CHANGE;
			END_IF

		PREVIEW_CHANGE:
			//Load a second time to ensure correct preview on page up/page down
			MpRecipe_0.Load := TRUE;
			HmiRecipe.Status.PreviewCase := PREVIEW_WAIT;

	END_CASE;

	// Reset load command on MpRecipe_0 FUB
	IF MpRecipe_0.StatusID <> 0 THEN
		HmiRecipe.Status.InvalidRecipe := TRUE;
		HmiRecipe.Commands.ResetPreview := TRUE;
	END_IF;

	IF ((MpRecipe_0.CommandDone = TRUE) OR (MpRecipe_0.Error = TRUE)) THEN
		MpRecipe_0.Load := FALSE;
	END_IF

END_ACTION

ACTION RecipeHMIcommands:

	CASE HmiRecipe.Status.HMIcommand OF
		REC_HMI_WAIT:
			// The following commands are triggered directly from the HMI. If you imported the mapp View front end of
			// the Framework, then this is already taken care of. If you did not, then your visualization must
			// trigger each one of these command variables (CreateRecipe, SaveSelectedRecipe, LoadRecipe).
			IF (MpRecipeUIConnect.Status <> mpRECIPE_UI_STATUS_IDLE) THEN
				// MpRecipe is active so don't issue a new command
			ELSIF HmiRecipe.Commands.CreateRecipe THEN
				HmiRecipe.Status.HMIcommand := REC_HMI_CREATE;
				HmiRecipe.Commands.CreateRecipe := FALSE;
			ELSIF HmiRecipe.Commands.SaveSelectedRecipe THEN
				HmiRecipe.Status.HMIcommand := REC_HMI_SAVE;
				HmiRecipe.Commands.SaveSelectedRecipe := FALSE;
			ELSIF HmiRecipe.Commands.LoadRecipe THEN
				HmiRecipe.Status.HMIcommand := REC_HMI_LOAD;
				HmiRecipe.Commands.LoadRecipe := FALSE;
				IF (brsstrcmp(ADR(HmiRecipe.Parameters.Category), ADR(PARAMETERS_RECIPE)) = 0) THEN
					HmiRecipe.Status.ProductRecipeLoaded := FALSE;
				ELSE
					HmiRecipe.Status.ConfigRecipeLoaded := FALSE;
				END_IF
			ELSIF HmiRecipe.Commands.ResetPreview THEN
				HmiRecipe.Status.HMIcommand := REC_HMI_RESET_PREVIEW;
				HmiRecipe.Commands.ResetPreview := FALSE;
			END_IF

		REC_HMI_CREATE:
			IF (brsstrcmp(ADR(HmiRecipe.Parameters.Category), ADR(PARAMETERS_RECIPE)) = 0) THEN
				ParametersPreview := ParametersEdit;
				brsstrcpy(ADR(MpRecipeUIConnect.New.FileName), ADR(HmiRecipe.Parameters.FileName));
				brsstrcat(ADR(MpRecipeUIConnect.New.FileName), ADR('.par'));
				// If the default recipe was initially missing and just now created, immediately load it
				IF HmiRecipe.Status.ParameterRecipeMissing THEN
					HmiRecipe.Commands.LoadRecipe := TRUE;
				END_IF
			ELSIF (brsstrcmp(ADR(HmiRecipe.Parameters.Category), ADR(MACHINE_CONFIGURATION_RECIPE)) = 0) THEN
				MachineSettingsPreview := MachineSettingsEdit;
				brsstrcpy(ADR(MpRecipeUIConnect.New.FileName), ADR(HmiRecipe.Parameters.FileName));
				brsstrcat(ADR(MpRecipeUIConnect.New.FileName), ADR('.mcfg'));
				// If the default recipe was initially missing and just now created, immediately load it
				IF HmiRecipe.Status.MachineSettingsRecipeMissing THEN
					HmiRecipe.Commands.LoadRecipe := TRUE;
				END_IF
			END_IF

			Header.Name := MpRecipeUIConnect.New.FileName;
			DTGetTime_0.enable := TRUE;
			REPEAT
				DTGetTime_0();
				UNTIL (DTGetTime_0.status = 0)
			END_REPEAT;
			Header.DateTime := DTGetTime_0.DT1;
			DTGetTime_0.enable := FALSE;
			DTGetTime_0();
			MpRecipeUIConnect.New.Create := TRUE;

			HmiRecipe.Status.HMIcommand := REC_HMI_WAIT;

		REC_HMI_LOAD:
			IF (MpRecipeUIConnect.Status = mpRECIPE_UI_STATUS_IDLE) THEN
				IF (brsstrcmp(ADR(HmiRecipe.Parameters.Category), ADR(PARAMETERS_RECIPE)) = 0) THEN
					Parameters := ParametersPreview;
					HmiRecipe.Status.ProductRecipeLoaded := TRUE;
					// If the default recipe was initially missing and just now created, then it is the last loaded recipe
					IF HmiRecipe.Status.ParameterRecipeMissing THEN
						HmiRecipe.Status.LastLoadedProductRecipe := DEFAULT_PARAMETERS;
						brsstrcat(ADR(HmiRecipe.Status.LastLoadedProductRecipe), ADR(PARAMETERS_FILE_EXTENSION));
						HmiRecipe.Status.ParameterRecipeMissing := FALSE;
						// Otherwise, the last loaded recipe is the selected recipe
					ELSE
						HmiRecipe.Status.LastLoadedProductRecipe := MpRecipeUIConnect.Recipe.List.Names[MpRecipeUIConnect.Recipe.List.SelectedIndex];
						HmiRecipeRetain.LastLoadedProductRecipe := MpRecipeUIConnect.Recipe.List.Names[MpRecipeUIConnect.Recipe.List.SelectedIndex];
					END_IF
				ELSIF (brsstrcmp(ADR(HmiRecipe.Parameters.Category), ADR(MACHINE_CONFIGURATION_RECIPE)) = 0) THEN
					MachineSettings := MachineSettingsPreview;
					HmiRecipe.Status.ConfigRecipeLoaded := TRUE;
					// If the default recipe was initially missing and just now created, then it is the last loaded recipe
					IF HmiRecipe.Status.MachineSettingsRecipeMissing THEN
						HmiRecipe.Status.LastLoadedConfigRecipe := DEFAULT_MACHINE_CONFIGURATION;
						brsstrcat(ADR(HmiRecipe.Status.LastLoadedConfigRecipe), ADR(MACHINE_CONFIG_FILE_EXTENSION));
						HmiRecipe.Status.MachineSettingsRecipeMissing := FALSE;
						// Otherwise, the last loaded recipe is the selected recipe
					ELSE
						HmiRecipe.Status.LastLoadedConfigRecipe := MpRecipeUIConnect.Recipe.List.Names[MpRecipeUIConnect.Recipe.List.SelectedIndex];
						HmiRecipeRetain.LastLoadedConfigRecipe := MpRecipeUIConnect.Recipe.List.Names[MpRecipeUIConnect.Recipe.List.SelectedIndex];
					END_IF
				END_IF
				HmiRecipe.Status.HMIcommand := REC_HMI_WAIT;
			END_IF

		REC_HMI_SAVE:
			IF (MpRecipeUIConnect.Status = mpRECIPE_UI_STATUS_IDLE) THEN

				IF (brsstrcmp(ADR(HmiRecipe.Parameters.Category), ADR(PARAMETERS_RECIPE)) = 0) THEN
					ParametersPreview := ParametersEdit;
				ELSIF (brsstrcmp(ADR(HmiRecipe.Parameters.Category), ADR(MACHINE_CONFIGURATION_RECIPE)) = 0) THEN
					MachineSettingsPreview := MachineSettingsEdit;
				END_IF

				IF (brsstrlen(ADR(HmiRecipe.Status.SelectedRecipe)) > 0) THEN
					MpRecipe_0.FileName := ADR(HmiRecipe.Status.SelectedRecipe);
					MpRecipe_0.Save := TRUE;
				END_IF

				HmiRecipe.Status.HMIcommand := REC_HMI_WAIT;
			END_IF

		REC_HMI_RESET_PREVIEW:
			IF (brsstrcmp(ADR(HmiRecipe.Parameters.Category), ADR(PARAMETERS_RECIPE)) = 0) THEN
				brsmemset(ADR(ParametersPreview), 0, SIZEOF(ParametersPreview));
			ELSIF (brsstrcmp(ADR(HmiRecipe.Parameters.Category), ADR(MACHINE_CONFIGURATION_RECIPE)) = 0) THEN
				brsmemset(ADR(MachineSettingsPreview), 0, SIZEOF(MachineSettingsPreview));
			END_IF
			HmiRecipe.Status.HMIcommand := REC_HMI_WAIT;

	END_CASE

	//	IF NOT MpRecipe_0.CommandBusy AND brsstrcmp(ADR(HmiRecipe.Status.PreviousRecipe), ADR(HmiRecipe.Parameters.FileName)) <> 0 THEN
	//		HmiRecipe.Parameters.FileName := HmiRecipe.Status.PreviousRecipe;
	//	END_IF

	// If the Edit or Create dialog boxes open, copy the Preview structure into the Edit structure.
	IF HmiRecipe.Status.EditDialogOpened OR HmiRecipe.Status.CreateDialogOpened THEN
		IF (brsstrcmp(ADR(HmiRecipe.Parameters.Category), ADR(PARAMETERS_RECIPE)) = 0) THEN
			ParametersEdit := ParametersPreview;
			IF HmiRecipe.Status.ParameterRecipeMissing THEN
				HmiRecipe.Parameters.FileName := DEFAULT_PARAMETERS;
			ELSE
				HmiRecipe.Parameters.FileName:= 'newParameters';
			END_IF
		ELSIF (brsstrcmp(ADR(HmiRecipe.Parameters.Category), ADR(MACHINE_CONFIGURATION_RECIPE)) = 0) THEN
			MachineSettingsEdit := MachineSettingsPreview;
			IF HmiRecipe.Status.MachineSettingsRecipeMissing THEN
				HmiRecipe.Parameters.FileName := DEFAULT_MACHINE_CONFIGURATION;
			ELSE
				HmiRecipe.Parameters.FileName := 'newMachineConfig';
			END_IF
		END_IF
		HmiRecipe.Status.EditDialogOpened := FALSE;
		HmiRecipe.Status.CreateDialogOpened := FALSE;
	END_IF

	// Check if the file name has already been used
	HmiRecipe.Status.FileDuplicate := FALSE;
	FOR i:=0 TO ((SIZEOF(MpRecipeUIConnect.Recipe.List.Names) / SIZEOF(MpRecipeUIConnect.Recipe.List.Names[0])) - 1) DO
		temp := HmiRecipe.Parameters.FileName;
		IF (brsstrcmp(ADR(HmiRecipe.Parameters.Category), ADR(PARAMETERS_RECIPE)) = 0) THEN
			brsstrcat(ADR(temp),ADR(PARAMETERS_FILE_EXTENSION));
		ELSIF (brsstrcmp(ADR(HmiRecipe.Parameters.Category), ADR(MACHINE_CONFIGURATION_RECIPE)) = 0) THEN
			brsstrcat(ADR(temp),ADR(MACHINE_CONFIG_FILE_EXTENSION));
		END_IF
		IF temp = MpRecipeUIConnect.Recipe.List.Names[i] THEN
			HmiRecipe.Status.FileDuplicate := TRUE;
		END_IF
	END_FOR

	// Set whether the loading .gif should be shown on the HMI
	HmiRecipe.Status.LoadingRecipeList := (MpRecipeUIConnect.Status = mpRECIPE_UI_STATUS_REFRESH);
	HmiRecipe.Status.DefaultRecipeSelected := (HmiRecipe.Status.SelectedRecipe = CONCAT(DEFAULT_PARAMETERS,PARAMETERS_FILE_EXTENSION)) OR (HmiRecipe.Status.SelectedRecipe = CONCAT(DEFAULT_MACHINE_CONFIGURATION, MACHINE_CONFIG_FILE_EXTENSION));

	// Update status information
	HmiRecipe.Status.LastStatus := MpRecipeUIConnect.Status;
	HmiRecipe.Status.SelectedRecipe := MpRecipeUIConnect.Recipe.List.Names[MpRecipeUIConnect.Recipe.List.SelectedIndex];

END_ACTION
```

#### RecipeMgr.st
```iecst
//***********************************************************************
// Copyright: B&R Industrial Automation GmbH
// Author: B&R Industrial Automation GmbH
// Created: Jan 1, 2022
// Description: Tasks for recipe control.
//***********************************************************************

PROGRAM _INIT

	// Create folder for this component on the user file device
	DirCreate_0(enable := TRUE, pDevice := ADR('mappRecipeFiles'), pName := ADR('/'));

	// Wait for DirCreate_0 to complete.
	WHILE (DirCreate_0.status = ERR_FUB_BUSY) DO
		DirCreate_0();
	END_WHILE

	// Check if folder already exist and if so disabled the function block call
	IF DirCreate_0.status = fiERR_DIR_ALREADY_EXIST OR (DirCreate_0.status = ERR_OK) THEN
		DirCreate_0(enable := FALSE);
	END_IF

	// Initialize mapp function blocks
	// By default, the Framework sets up an XML recipe system. To swtich to the CSV format, refer to the "Change Recipe Format"
	// page in the AS Help (GUID 2052b3a5-f59b-45f9-9fcd-3289c93401af)
	MpRecipeUISetup.Confirmation.RecipeDelete := TRUE;
	MpRecipeUISetup.RecipeListSize := 9;
	MpRecipeUISetup.RecipeListScrollWindow := 0;
	MpRecipeUISetup.AutoLoadHeader := TRUE;
	MpRecipeUIConnect.New.FileName := 'newRecipe';
	MpRecipeUIConnect.Recipe.Filter := '*par';
	MpRecipeUI_0.MpLink := ADR(gMpLinkRecipeXml);
	MpRecipeUI_0.Enable := TRUE;
	MpRecipeUI_0.UIConnect := ADR(MpRecipeUIConnect);
	MpRecipeUI_0.UISetup := MpRecipeUISetup;
	MpRecipeUI_0();

	HmiRecipe.Parameters.Category := PARAMETERS_CATEGORY;
	HmiRecipe.Status.DeviceDataProvider[0] := '{"value":"mappRecipeFiles","text":"CF/PLC"}';
	HmiRecipe.Parameters.DeviceName := 'mappRecipeFiles';
	MpRecipe_0.MpLink := ADR(gMpLinkRecipeXml);
	MpRecipe_0.Enable := TRUE;
	MpRecipe_0.Category := ADR(HmiRecipe.Parameters.Category);
	MpRecipe_0.DeviceName := ADR(HmiRecipe.Parameters.DeviceName);
	MpRecipe_0.FileName := ADR(HmiRecipe.Parameters.FileName);
	MpRecipe_0.Header := ADR(Header);

	// Wait for MpRecipe_0 to activate. This must be active before you can call the RegPar function blocks, which is below.
	WHILE NOT(MpRecipe_0.Active OR MpRecipe_0.Error) DO
		MpRecipe_0();
	END_WHILE

	// Register the preview variables to the recipe. These preview variables are a buffer between the recipe system and the
	// variables used at runtime on the machine (Parameters, MachineSettings). By using these preview variables, you can
	// preview and edit a recipe on the HMI without actually loading it to the machine. For more details, refer to the
	// "Recipe System Design" page in the AS Help (GUID 3ccd7409-0b52-4bbc-a93a-4010f6db414c).

	MpRecipeRegPar_PreviewPar.MpLink := ADR(gMpLinkRecipeXml);
	MpRecipeRegPar_PreviewPar.Enable := TRUE;
	MpRecipeRegPar_PreviewPar.PVName := ADR('RecipeMgr:ParametersPreview');
	MpRecipeRegPar_PreviewPar.Category := ADR(PARAMETERS_CATEGORY);
	MpRecipeRegPar_PreviewPar();

	MpRecipeRegPar_PreviewCfg.MpLink := ADR(gMpLinkRecipeXml);
	MpRecipeRegPar_PreviewCfg.Enable := TRUE;
	MpRecipeRegPar_PreviewCfg.PVName := ADR('RecipeMgr:MachineSettingsPreview');
	MpRecipeRegPar_PreviewCfg.Category := ADR(MACHINE_CONFIGURATION_CATEGORY);
	MpRecipeRegPar_PreviewCfg();

	// Wait for RegPar function blocks to activate. These must be active before you can load a recipe,
	// which is further down in the Initialization program.
	WHILE NOT(MpRecipeRegPar_PreviewPar.Active OR MpRecipeRegPar_PreviewPar.Error) DO
		MpRecipeRegPar_PreviewPar();
	END_WHILE
	WHILE NOT(MpRecipeRegPar_PreviewCfg.Active OR MpRecipeRegPar_PreviewCfg.Error) DO
		MpRecipeRegPar_PreviewCfg();
	END_WHILE

	// Load default Machine Settings recipe
	HmiRecipe.Parameters.Category := MACHINE_CONFIGURATION_CATEGORY;
	IF (brsstrcmp(ADR(HmiRecipeRetain.LastLoadedConfigRecipe), ADR('')) <> 0) THEN
		HmiRecipe.Parameters.FileName := HmiRecipeRetain.LastLoadedConfigRecipe;
	ELSE
		HmiRecipe.Parameters.FileName := DEFAULT_MACHINE_CONFIGURATION;
		brsstrcat(ADR(HmiRecipe.Parameters.FileName),ADR(MACHINE_CONFIG_FILE_EXTENSION));
	END_IF
	MpRecipe_0.Load := TRUE;
	WHILE NOT(MpRecipe_0.CommandDone OR MpRecipe_0.Error) DO
		MpRecipe_0();
	END_WHILE
	MachineSettings := MachineSettingsPreview;
	IF (brsstrcmp(ADR(HmiRecipeRetain.LastLoadedConfigRecipe), ADR('')) <> 0) THEN
		HmiRecipe.Status.LastLoadedConfigRecipe := HmiRecipeRetain.LastLoadedConfigRecipe;
	ELSE
		HmiRecipe.Status.LastLoadedConfigRecipe := DEFAULT_MACHINE_CONFIGURATION;
		brsstrcat(ADR(HmiRecipe.Status.LastLoadedConfigRecipe),ADR(MACHINE_CONFIG_FILE_EXTENSION));
		HmiRecipeRetain.LastLoadedConfigRecipe := HmiRecipe.Status.LastLoadedConfigRecipe;
	END_IF
	HmiRecipe.Status.ConfigRecipeLoaded := TRUE;

	// Check if the default machine settings recipe is missing
	IF MpRecipe_0.Info.Diag.StatusID.ID = mpRECIPE_ERR_LOAD_DATA THEN
		HmiRecipe.Status.MachineSettingsRecipeMissing := TRUE;
		HmiRecipe.Status.LastLoadedConfigRecipe := '';
		HmiRecipe.Status.ConfigRecipeLoaded := FALSE;
	END_IF

	MpRecipe_0.ErrorReset := MpRecipe_0.Error;
	MpRecipe_0.Load := FALSE;
	MpRecipe_0();

	// Load default Parameter recipe
	HmiRecipe.Parameters.Category := PARAMETERS_CATEGORY;
	IF (brsstrcmp(ADR(HmiRecipeRetain.LastLoadedProductRecipe), ADR('')) <> 0) THEN
		HmiRecipe.Parameters.FileName := HmiRecipeRetain.LastLoadedProductRecipe;
	ELSE
		HmiRecipe.Parameters.FileName := DEFAULT_PARAMETERS;
		brsstrcat(ADR(HmiRecipe.Parameters.FileName),ADR(PARAMETERS_FILE_EXTENSION));
	END_IF
	HmiRecipe.Status.PreviousRecipe := DEFAULT_PARAMETERS;
	MpRecipe_0.Load := TRUE;
	WHILE NOT(MpRecipe_0.CommandDone OR MpRecipe_0.Error) DO
		MpRecipe_0();
	END_WHILE
	Parameters := ParametersPreview;
	IF (brsstrcmp(ADR(HmiRecipeRetain.LastLoadedProductRecipe), ADR('')) <> 0) THEN
		HmiRecipe.Status.LastLoadedProductRecipe := HmiRecipeRetain.LastLoadedProductRecipe;
	ELSE
		HmiRecipe.Status.LastLoadedProductRecipe := DEFAULT_PARAMETERS;
		brsstrcat(ADR(HmiRecipe.Status.LastLoadedProductRecipe),ADR(PARAMETERS_FILE_EXTENSION));
		HmiRecipeRetain.LastLoadedProductRecipe := HmiRecipe.Status.LastLoadedProductRecipe;
	END_IF
	HmiRecipe.Status.ProductRecipeLoaded := TRUE;

	// Check if the default parameters recipe is missing
	IF MpRecipe_0.Info.Diag.StatusID.ID = mpRECIPE_ERR_LOAD_DATA THEN
		HmiRecipe.Status.ParameterRecipeMissing := TRUE;
		HmiRecipe.Status.LastLoadedProductRecipe := '';
		HmiRecipe.Status.ProductRecipeLoaded := FALSE;
	END_IF

	MpRecipe_0.ErrorReset := MpRecipe_0.Error;
	MpRecipe_0.Load := FALSE;
	MpRecipe_0();

	// Trigger update notification so that the initial parameters are copied to the process
	MpRecipe_0.UpdateNotification := TRUE;

	// Init Filemanager for exporting/importing files
	MpFileManagerUI_0.Enable := TRUE;
	MpFileManagerUI_0.MpLink := ADR(gMpLinkFileManagerUIRecipe);
	MpFileManagerUI_0.UIConnect := ADR(MpFileManagerUIConnect);
	MpFileManagerUI_0.UISetup.FileListSize := SIZEOF(MpFileManagerUIConnect.File.List.Items) / SIZEOF(MpFileManagerUIConnect.File.List.Items[0]);
	MpFileManagerUIConnect.DeviceList.DeviceNames[0] := 'mappRecipeFiles';
	MpFileManagerUIConnect.DeviceList.DeviceNames[1] := '';
	MpFileManagerUI_0();

	HmiRecipe.Status.HMIcommand := REC_HMI_WAIT;

END_PROGRAM

PROGRAM _CYCLIC

	// Call all cyclic actions
	FormatDeviceDataProvider;
	LoadPreview;
	RecipeHMIcommands;
	LoadStatus;

	// Reset commands on MpRecipe FUB
	IF MpRecipe_0.CommandDone THEN
		MpRecipe_0.Load := FALSE;
		MpRecipe_0.Save := FALSE;
		// Set update notification for machine category
		IF ((brsstrcmp(ADR(HmiRecipe.Parameters.Category), ADR(MACHINE_CONFIGURATION_CATEGORY)) = 0) AND (MpRecipe_0.Save = TRUE)) THEN
			MpRecipe_0.UpdateNotification := TRUE;
		ELSE
			MpRecipe_0.UpdateNotification := FALSE;
		END_IF
	END_IF

	// Error reset
	IF NOT MpRecipe_0.Error THEN
		MpRecipe_0.ErrorReset := FALSE;
	END_IF

	IF NOT MpRecipeUI_0.Error THEN
		MpRecipeUI_0.ErrorReset := FALSE;
	END_IF

	// Assign MpLinks & address references
	MpRecipe_0.MpLink := ADR(gMpLinkRecipeXml);
	MpRecipe_0.DeviceName := ADR(HmiRecipe.Parameters.DeviceName);
	MpRecipe_0.Header := ADR(Header);
	MpRecipeUI_0.MpLink := ADR(gMpLinkRecipeXml);
	MpRecipeUI_0.UIConnect := ADR(MpRecipeUIConnect);
	MpFileManagerUI_0.MpLink := ADR(gMpLinkFileManagerUIRecipe);
	MpRecipeRegPar_PreviewPar.MpLink := ADR(gMpLinkRecipeXml);
	MpRecipeRegPar_PreviewPar.PVName := ADR('RecipeMgr:ParametersPreview');
	MpRecipeRegPar_PreviewPar.Category := ADR(PARAMETERS_CATEGORY);
	MpRecipeRegPar_PreviewCfg.MpLink := ADR(gMpLinkRecipeXml);
	MpRecipeRegPar_PreviewCfg.PVName := ADR('RecipeMgr:MachineSettingsPreview');
	MpRecipeRegPar_PreviewCfg.Category := ADR(MACHINE_CONFIGURATION_CATEGORY);
	MpFileManagerUI_0.UIConnect := ADR(MpFileManagerUIConnect);

	// Call function blocks
	MpRecipe_0();
	MpRecipeUI_0();
	MpFileManagerUI_0();
	MpRecipeRegPar_PreviewPar();
	MpRecipeRegPar_PreviewCfg();

END_PROGRAM

PROGRAM _EXIT

	// Disable the function blocls to unlink the MpLinks
	MpRecipe_0.Enable := FALSE;
	MpRecipeUI_0.Enable := FALSE;
	MpRecipeRegPar_PreviewPar.Enable := FALSE;
	MpRecipeRegPar_PreviewCfg.Enable := FALSE;
	MpFileManagerUI_0.Enable := FALSE;

	// Call function blocks
	MpRecipe_0();
	MpRecipeUI_0();
	MpRecipeRegPar_PreviewPar();
	MpRecipeRegPar_PreviewCfg();
	MpFileManagerUI_0();

END_PROGRAM
```

### Package Logical/Infrastructure/UserX - Package for mapp UserX Framework

### Program Logical/Infrastructure/UserX/UserXMgr (IEC)

#### UserXMgr.st - Init, cyclic, exit code
```iecst
//***********************************************************************
// Copyright: B&R Industrial Automation GmbH
// Author: B&R Industrial Automation GmbH
// Created: April 12, 2022
// Description: Tasks for user management.
//***********************************************************************

PROGRAM _INIT

	// Create folder for this component on the user file device
	DirCreate_0(enable := TRUE, pDevice := ADR('mappUserXFiles'), pName := ADR('/'));

	// Check if folder already exist and if so disabled the function block call
	IF DirCreate_0.status = fiERR_DIR_ALREADY_EXIST THEN
		DirCreate_0(enable := FALSE);
	END_IF

	// Initialize mapp function blocks
	UserXMgrUIConnect.User.Create.Lock := FALSE;
	UserXMgrUIConnect.User.Lock := FALSE;
	UserXMgrUIConnect.User.Edit.Lock := FALSE;
	UserXMgrUIConnect.User.Create.Dialog.UserName := "";
	UserXMgrUIConnect.User.Create.Dialog.NewPassword := "";
	UserXMgrUIConnect.User.Create.Dialog.ConfirmPassword := "";
	UserXMgrUIConnect.User.List.MaxSelection := USER_LIST_MAX_SELECTION;
	UserXMgrUIConnect.User.List.RangeStart := USER_LIST_RANGE_START;
	UserXMgrUIConnect.User.List.RangeEnd := USER_LIST_RANGE_END;
	MpUserXManagerUI_0.MpLink := ADR(gMpLinkUserXLogin);
	MpUserXManagerUI_0.Enable := TRUE;
	MpUserXManagerUI_0.UIConnect := ADR(UserXMgrUIConnect);
	MpUserXManagerUI_0();

	MpUserXLoginUI_0.MpLink := ADR(gMpLinkUserXLogin);
	MpUserXLoginUI_0.Enable := TRUE;
	MpUserXLoginUI_0.UIConnect := ADR(UserXLoginUIConnect);
	MpUserXLoginUI_0();

	MpUserXLogin_0.MpLink := ADR(gMpLinkUserXLogin);
	MpUserXLogin_0.Enable := TRUE;
	MpUserXLogin_0();

END_PROGRAM

PROGRAM _CYCLIC

	// Error reset
	IF NOT MpUserXManagerUI_0.Error THEN
		MpUserXManagerUI_0.ErrorReset := FALSE;
	END_IF

	IF NOT MpUserXLoginUI_0.Error THEN
		MpUserXLoginUI_0.ErrorReset := FALSE;
	END_IF

	IF NOT MpUserXLogin_0.Error THEN
		MpUserXLogin_0.ErrorReset := FALSE;
	END_IF

	// Call all cyclic actions
	HMIAction;

	// Saving last status of UserXMgrUIconnect
	HmiUserX.Status.LastMgrConnectStatus := UserXMgrUIConnect.Status;

	// Assign MpLinks & address references
	MpUserXManagerUI_0.MpLink := ADR(gMpLinkUserXLogin);
	MpUserXManagerUI_0.UIConnect := ADR(UserXMgrUIConnect);
	MpUserXLoginUI_0.MpLink := ADR(gMpLinkUserXLogin);
	MpUserXLoginUI_0.UIConnect := ADR(UserXLoginUIConnect);
	MpUserXLogin_0.MpLink := ADR(gMpLinkUserXLogin);

	// Call function blocks
	MpUserXManagerUI_0();
	MpUserXLoginUI_0();
	MpUserXLogin_0();

END_PROGRAM

PROGRAM _EXIT

	// Disable the function blocls to unlink the MpLinks
	MpUserXManagerUI_0.Enable := FALSE;
	MpUserXLoginUI_0.Enable := FALSE;
	MpUserXLogin_0.Enable := FALSE;

	// Call function blocks
	MpUserXManagerUI_0();
	MpUserXLoginUI_0();
	MpUserXLogin_0();

END_PROGRAM
```

#### UserXMgr.typ - Local data types
```iecst
(*Structure types*)

TYPE
	UserXHmiInterfaceType : 	STRUCT  (*Structure to hold commands and status from the HMI*)
		Commands : UserXCommandsType; (*Structure to hold the commands from the HMI*)
		Status : UserXStatusType; (*Structure to hold status information to the HMI*)
	END_STRUCT;
	UserXCommandsType : 	STRUCT  (*Structure to hold the commands from the HMI*)
		Export : BOOL; (*Export a user list*)
		ConfirmOverwrite : BOOL; (*Confirm you want to overwrite an existing user export with the same filenmae*)
	END_STRUCT;
	UserXStatusType : 	STRUCT  (*Structure to hold status information to the HMI*)
		FileDuplicate : BOOL; (*Flag that a user export file already exists with the specified name*)
		UserXHmiState : HmiStateEnum; (*State variable for HMI interaction*)
		LastMgrConnectStatus : MpUserXUIStatusEnum;
		ExportComplete : BOOL;
		UserExportDisplayed : BOOL;
	END_STRUCT;
END_TYPE

(*Enumerations*)

TYPE
	HmiStateEnum :
		( (*State enumeration for HMI interaction*)
		USERX_START := 0,
		USERX_WAIT_FOR_DIALOG := 1,
		USERX_SET_RESPONSE := 2,
		USERX_CONFIRM_RESPONSE := 3,
		USERX_NEW_EXPORT := 4,
		USERX_FINISH := 5
		);
END_TYPE
```

#### UserXMgr.var - Local variables
```iecst
(*Function Blocks*)
VAR
	MpUserXLogin_0 : MpUserXLogin; (*MpUserXLogin instance*)
	MpUserXManagerUI_0 : MpUserXManagerUI := (UISetup:=(FileDevice:='mappUserXFiles')); (*MpUserXManagerUI instance*)
	MpUserXLoginUI_0 : MpUserXLoginUI; (*MpUserXLoginUI instance*)
	DirCreate_0 : DirCreate; (*DirCreate instance*)
END_VAR
(*Constants*)
VAR CONSTANT
	USER_LIST_MAX_SELECTION : USINT := 20; (*Maxiumum selections on the User List *)
	USER_LIST_RANGE_START : USINT := 0; (*Range start (used for UserXMgrUIConnect)*)
	USER_LIST_RANGE_END : USINT := 20; (*Range end (used for UserXMgrUIConnect)*)
END_VAR
(*Structure Types*)
VAR
	UserXMgrUIConnect : MpUserXMgrUIConnectType; (*UserX manager connection to the HMI*)
	UserXLoginUIConnect : MpUserXLoginUIConnectType; (*UserL login connection to the HMI*)
	HmiUserX : UserXHmiInterfaceType; (*HMI interface structure *)
END_VAR
(*Variables*)
VAR
	temp : STRING[255]; (*Temporary string holder for checking file names*)
	i : USINT; (*Index*)
END_VAR
(*Enumerations*)
```

#### HMIAction.st
```iecst
ACTION HMIAction:
	CASE HmiUserX.Status.UserXHmiState OF
		USERX_START:
			IF NOT UserXMgrUIConnect.Import.ShowDialog THEN
				UserXMgrUIConnect.Import.ShowDialog := TRUE;
			ELSE
				HmiUserX.Status.UserXHmiState := USERX_WAIT_FOR_DIALOG;
			END_IF
		USERX_WAIT_FOR_DIALOG:
			UserXMgrUIConnect.Import.ShowDialog := FALSE;
			HmiUserX.Status.UserXHmiState := USERX_SET_RESPONSE;
		USERX_SET_RESPONSE:
			IF NOT(UserXMgrUIConnect.Status = mpUSERX_UI_STATUS_IDLE) THEN
				UserXMgrUIConnect.Import.Dialog.Cancel := TRUE;
			ELSE
				UserXMgrUIConnect.Import.Dialog.Cancel := FALSE;
				HmiUserX.Status.UserXHmiState := USERX_CONFIRM_RESPONSE;
			END_IF
		USERX_CONFIRM_RESPONSE:
			IF UserXMgrUIConnect.Status = mpUSERX_UI_STATUS_WAIT_DLG THEN
				HmiUserX.Status.UserXHmiState := USERX_START;
			ELSE
				HmiUserX.Status.UserXHmiState := USERX_FINISH;
			END_IF
		USERX_NEW_EXPORT:
			IF NOT UserXMgrUIConnect.Export.ShowDialog AND UserXMgrUIConnect.Status = mpUSERX_UI_STATUS_IDLE THEN
				HmiUserX.Status.UserXHmiState := USERX_START;
			END_IF
		USERX_FINISH:

	END_CASE
	// If new updates are made via export execute a check
	IF UserXMgrUIConnect.Export.ShowDialog THEN
		HmiUserX.Status.UserXHmiState := USERX_NEW_EXPORT;
	END_IF

	// Duplicate file checks
	HmiUserX.Status.FileDuplicate := FALSE;
	FOR i := 0 TO ((SIZEOF(UserXMgrUIConnect.Import.Dialog.List.FileNames) / SIZEOF(UserXMgrUIConnect.Import.Dialog.List.FileNames[0])) - 1) DO
		temp := UserXMgrUIConnect.Export.Dialog.FileName;
		brsstrcat(ADR(temp),ADR('.usr'));
		IF (temp = UserXMgrUIConnect.Import.Dialog.List.FileNames[i]) AND HmiUserX.Commands.Export THEN
			HmiUserX.Status.FileDuplicate := TRUE;
		END_IF
	END_FOR

	IF HmiUserX.Status.FileDuplicate AND (HmiUserX.Commands.ConfirmOverwrite) THEN
		UserXMgrUIConnect.Export.Dialog.Confirm := TRUE;
		HmiUserX.Commands.Export := FALSE;
		HmiUserX.Commands.ConfirmOverwrite := FALSE;
	ELSIF NOT HmiUserX.Status.FileDuplicate AND HmiUserX.Commands.Export THEN
		UserXMgrUIConnect.Export.Dialog.Confirm := TRUE;
		HmiUserX.Commands.Export := FALSE;
	END_IF

	// Export confirmation pop-up handling
	IF (HmiUserX.Status.LastMgrConnectStatus = mpUSERX_UI_STATUS_WAIT_DLG) AND (UserXMgrUIConnect.Status = mpUSERX_UI_STATUS_IDLE) AND UserXMgrUIConnect.Export.Dialog.Confirm THEN
		HmiUserX.Status.ExportComplete := TRUE;
	END_IF

	IF HmiUserX.Status.UserExportDisplayed THEN
		HmiUserX.Status.ExportComplete := FALSE;
		HmiUserX.Status.UserExportDisplayed := FALSE;
		UserXMgrUIConnect.Export.Dialog.Confirm := FALSE;
	END_IF

END_ACTION
```

### Package Logical/Infrastructure/Audit - Package for mapp Audit Framework

### Program Logical/Infrastructure/Audit/AuditMgr (IEC) - Audit manager

#### AuditMgr.st - Init, cyclic, exit code
```iecst
//***********************************************************************
// Copyright: B&R Industrial Automation GmbH
// Author: B&R Industrial Automation GmbH
// Created: Sept 1, 2022
// Description: Task for audit management.
//***********************************************************************

PROGRAM _INIT

	// Create folder for this component on the user file device
	DirCreate_0(enable := TRUE, pDevice := ADR('mappAuditFiles'), pName := ADR('/'));

	// Check if folder already exist and if so disabled the function block call
	IF DirCreate_0.status = fiERR_DIR_ALREADY_EXIST THEN
		DirCreate_0(enable := FALSE);
	END_IF

	// Initialize mapp function blocks
	MpAuditTrail_0.Enable := TRUE;
	MpAuditTrail_0.MpLink := ADR(gMpLinkAuditTrail);
	MpAuditTrail_0.Language := ADR('en');
	MpAuditTrail_0.DeviceName := ADR('mappAuditFiles');
	MpAuditTrail_0();

	MpAuditTrailConfig_0.Enable := TRUE;
	MpAuditTrailConfig_0.MpLink := ADR(gMpLinkAuditTrail);
	MpAuditTrailConfig_0.Configuration := ADR(AuditTrailConfig);
	MpAuditTrailConfig_0.Load := TRUE;
	MpAuditTrailConfig_0();

	MpAuditTrail_CEvents.Enable := TRUE;
	MpAuditTrail_CEvents.MpLink := ADR(gMpLinkCustomEvents);
	MpAuditTrail_CEvents();

	MpAuditTrailUI_0.MpLink := ADR(gMpLinkAuditTrail);
	MpAuditTrailUI_0.UIConnect := ADR(MpAuditTrailUIConnect);
	MpAuditTrailUI_0.UISetup.EventListSize := SIZEOF(MpAuditTrailUIConnect.Output.EventID) / SIZEOF(MpAuditTrailUIConnect.Output.EventID[0]);
	MpAuditTrailUI_0.UISetup.ScrollWindow := 1;
	MpAuditTrailUI_0.Enable := TRUE;
	MpAuditTrailUI_0();

	// Initialize custom events
	CustomEvent[0].Type := "Custom Event Type";
	CustomEvent[0].Msg := "Custom Event Message";
	CustomEvent[0].Comment := "Custom Event Comment";

	CustomEvent[1].Type := "Audit Test";
	CustomEvent[1].Msg := "This is a custom event test msg";
	CustomEvent[1].Comment := "If you see this it was a success!";

	CustomEvent[2].Type := "Cmd Exe";
	CustomEvent[2].Msg := "The run query command was pressed on the HMI";
	CustomEvent[2].Comment := "Result can be seen in the Query tab";

	HmiAudit.Status.Query.Name := 'UserEvents';
	HmiAudit.Status.Query.Option := 0;

	// Configuring the query selection, reading the available components
	HmiAudit.Parameters.QuerySelection[0] := 'UserXMgr';
	HmiAudit.Parameters.QuerySelection[1] := 'RecipeMgr';

	IF (ST_ident(ADR(HmiAudit.Parameters.QuerySelection[0]), 0, ADR(ident)) = 0) AND (ST_ident(ADR(HmiAudit.Parameters.QuerySelection[1]), 0, ADR(ident)) = 0) THEN
		HmiAudit.Status.DeviceDataProvider[0] := '{"value":"UserEvents","text":"User Events Query"}';
		HmiAudit.Status.DeviceDataProvider[1] := '{"value":"RecipeEvents","text":"Recipe Events Query"}';
	ELSIF (ST_ident(ADR(HmiAudit.Parameters.QuerySelection[0]), 0, ADR(ident)) <> 0) AND (ST_ident(ADR(HmiAudit.Parameters.QuerySelection[1]), 0, ADR(ident)) = 0) THEN
		HmiAudit.Status.DeviceDataProvider[0] := '{"value":"RecipeEvents","text":"Recipe Events Query"}';
	ELSIF (ST_ident(ADR(HmiAudit.Parameters.QuerySelection[0]), 0, ADR(ident)) = 0) AND (ST_ident(ADR(HmiAudit.Parameters.QuerySelection[1]), 0, ADR(ident)) <> 0) THEN
		HmiAudit.Status.DeviceDataProvider[0] := '{"value":"UserEvents","text":"User Events Query"}';
	END_IF

	// Restored the retained values to the archive settings
	HmiAudit.Parameters.ArchiveSettings := ArchiveSettingsRetain;

END_PROGRAM

PROGRAM _CYCLIC

	// Call all cyclic actions
	ExecuteQuery;
	QueryTableConfig;
	ArchiveExport;
	ArchiveSettings;
	ChangeConfiguration;

	// Sample code for how custom events can be triggered. Use custom events as needed around the application for debugging purposes.
	IF EDGEPOS(CustomEvent[0].Set) THEN
		MpAuditCustomEvent(gMpLinkCustomEvents,CustomEvent[0].Type,CustomEvent[0].Msg,CustomEvent[0].Comment);
	END_IF
	IF EDGENEG(CustomEvent[1].Set) THEN
		MpAuditCustomEvent(gMpLinkCustomEvents,CustomEvent[1].Type,CustomEvent[1].Msg,CustomEvent[1].Comment);
	END_IF

	// Change sample variable randomly to trigger a value change event
	IF VariableMonitorExample = 0 THEN
		VariableMonitorExample := 10.5;
	END_IF

	// Error reset
	IF NOT MpAuditTrail_0.Error THEN
		MpAuditTrail_0.ErrorReset := FALSE;
	END_IF

	// Assign MpLinks & address references
	MpAuditTrail_0.MpLink := ADR(gMpLinkAuditTrail);
	MpAuditTrail_0.DeviceName := ADR('mappAuditFiles');
	MpAuditTrailConfig_0.MpLink := ADR(gMpLinkAuditTrail);
	MpAuditTrailConfig_0.Configuration := ADR(AuditTrailConfig);
	MpAuditTrail_CEvents.MpLink := ADR(gMpLinkCustomEvents);
	MpAuditTrailUI_0.MpLink := ADR(gMpLinkAuditTrail);
	MpAuditTrailUI_0.UIConnect := ADR(MpAuditTrailUIConnect);

	// Call function blocks
	MpAuditTrail_0();
	MpAuditTrailConfig_0();
	MpAuditTrail_CEvents();
	MpAuditTrailUI_0();

END_PROGRAM

PROGRAM _EXIT

	// Disable the function blocks to unlink the MpLinks
	MpAuditTrail_0.Enable := FALSE;
	MpAuditTrailConfig_0.Enable := FALSE;
	MpAuditTrail_CEvents.Enable := FALSE;
	MpAuditTrailUI_0.Enable := FALSE;

	// Call function blocks
	MpAuditTrail_0();
	MpAuditTrailConfig_0();
	MpAuditTrail_CEvents();
	MpAuditTrailUI_0();

END_PROGRAM
```

#### AuditMgr.typ - Local data types
```iecst
(*Structure types*)

TYPE
	AuditQueryHMIType : 	STRUCT  (*Datatype for the structure which rearranges the query data from AuditQuery into a structure of arrays for easy connection to the Table widget in mapp View*)
		EvTime : ARRAY[0..MAX_QUERY_RESULTS]OF DATE_AND_TIME; (*ActiveAudits query, Event-Time column*)
		Text : ARRAY[0..MAX_QUERY_RESULTS]OF WSTRING[100]; (*ActiveAudits query, Text column*)
		DText : ARRAY[0..MAX_QUERY_RESULTS]OF WSTRING[100]; (*ActiveAudits query, Display Text column*)
		Op : ARRAY[0..MAX_QUERY_RESULTS]OF WSTRING[100]; (*ActiveAudits query, Operator-Name column*)
		QueryCount : USINT; (*Count of query results for building the query table configuration string*)
		Name : STRING[80]; (*Name of the query to be executed*)
		Option : USINT; (*Index value of the selected query type in the dropdown on the query tab*)
	END_STRUCT;
	AuditCustomEventType : 	STRUCT  (*Structure for custom events handling*)
		Set : BOOL; (*Trigger the assigned function*)
		Type : WSTRING[100]; (*Entered when creating the entry under %typ*)
		Msg : WSTRING[100]; (*Entered when creating the entry under %msg *)
		Comment : WSTRING[100]; (*Entered when creating the entry under %cmt *)
	END_STRUCT;
	AuditQueryType : 	STRUCT  (*Structure for query results and status*)
		State : ActiveAuditStateEnum; (*State variable for the query state machine*)
		LastUpdateCount : UDINT; (*Previous count of query results. Used to check for new query data. *)
		UpdateCountRecipe : UDINT; (*Count of query results. Increases each time new results are availble. *)
		UpdateCount : UDINT; (*Count of query results. Increases each time new results are availble. *)
		Audits : ARRAY[0..MAX_QUERY_RESULTS]OF AuditType; (*Query data*)
		Next : BOOL; (*Trigger to query the next data, if there are more results than MAX_QUERY_RESULTS*)
	END_STRUCT;
	AuditHmiInterfaceType : 	STRUCT  (*Structure to hold commands and status from the HMI*)
		Commands : AuditCommandsType; (*HMI commands*)
		Parameters : AuditParametersType; (*HMI parameters*)
		Status : {REDUND_UNREPLICABLE} AuditStatusType; (*HMI status*)
	END_STRUCT;
	AuditCommandsType : 	STRUCT  (*Structure to hold the commands from the HMI*)
		ExportArchives : BOOL; (*Triggers an Audit export of the Audit history. Connected to a button on the HMI. *)
		RunQuery : BOOL; (*Triggers the query to run. Connected to a button on the HMI. *)
		SaveConfig : BOOL; (*Starts the configuration for archives*)
	END_STRUCT;
	AuditStatusType : 	STRUCT  (*Structure to hold status information from the mapp View HMI. (This structure is not compatible/relevant if you are using a VC4 visualization)*)
		AuditSortCfg : STRING[1000]; (*Sort configuration for the AuditList widget*)
		AuditFilterCfg : STRING[1000]; (*Filter configuration for the AuditList widget*)
		TableConfig : ARRAY[0..1]OF STRING[255]; (*Table configuration for the Audit query Table*)
		Query : AuditQueryHMIType; (*Structure which rearranges the query data from AuditQuery into a structure of arrays for easy connection to the Table widget*)
		CustomEventSortCfg : STRING[1000]; (*Sort configuration for the AuditList Custom Events widget*)
		CustomEventsFilterCfg : STRING[1000]; (*Filter configuration for the AuditList Custom Events widget*)
		ArchiveAvailable : BOOL; (*At least 1 archive is available for export*)
		NumberOfArchives : UINT; (*How many archives are available for export*)
		DeviceDataProvider : ARRAY[0..1]OF STRING[100]; (*Data provider for the file device selector*)
	END_STRUCT;
	AuditParametersType : 	STRUCT  (*Structure to hold parameter data for the HMI*)
		ArchiveSettings : AuditArchiveParType; (*Parameter for archive configuration*)
		QuerySelection : ARRAY[0..MAX_QUERIES]OF STRING[10]; (*The selection in the query dropdown on the query tab of the Audit content*)
	END_STRUCT;
	AuditArchiveParType : 	STRUCT  (*Automatic archive settings*)
		Enable : BOOL; (*Enable automatic archive feature*)
		MaxSize : UDINT; (*Name prefix for each automatic backup file*)
		Mode : MpAuditArchiveModeEnum; (*Mode (daily, Mo-Fr or by batch)*)
		Hour : USINT; (*Time (hour)*)
		Minute : USINT; (*Time (minutes)*)
		FileType : MpAuditFileTypeEnum := mpAUDIT_FILE_TYPE_XML; (*File type selection (XML, TXT, PDF)*)
	END_STRUCT;
	AuditType : 	STRUCT  (*Structure to hold the Audit data for the query results*)
		EvTime : DATE_AND_TIME; (*ActiveAudits query, Event-Time column*)
		Text : WSTRING[100]; (*ActiveAudits query, Text column*)
		DText : WSTRING[100]; (*ActiveAudits query, Display Text column*)
		Op : WSTRING[100]; (*ActiveAudits query, Operator-Name column*)
	END_STRUCT;
END_TYPE

(*Enumerations*)

TYPE
	ActiveAuditStateEnum :
		( (*Enumeration for the state for the query state machine*)
		ACTIVE_AUDIT_WAIT, (*Wait state*)
		ACTIVE_AUDIT_QUERY, (*State to query the Audit data*)
		ACTIVE_AUDIT_NEXT (*State to check if more Audits meet the query criteria and need to be queried*)
		);
END_TYPE
```

#### AuditMgr.var - Local variables
```iecst
(*Function Blocks*)
VAR
	DirCreateAudit : DirCreate; (*DirCreate instance*)
	MpAuditTrailSys : MpAuditTrail; (*AuditTrail for regular mapp events*)
	MpAuditTrailConfigSys : MpAuditTrailConfig; (*AuditTrail configuration*)
	MpAuditTrailCEvents : MpAuditTrail; (*AuditTrail for custom events*)
	QueryUserEvents : {REDUND_UNREPLICABLE} MpAuditQuery; (*MpAlarmXQuery instance*)
	MpAuditTrailUISys : MpAuditTrailUI; (*AuditTrail UI interface*)
END_VAR
(*Constants*)
VAR CONSTANT
	MAX_QUERY_RESULTS : USINT := 19; (*Maximum number of query results (Value+1)*)
	MAX_CUSTOM_EVENTS : USINT := 9; (*Maximum number of custom events*)
	MAX_QUERIES : USINT := 2; (*Maximum number of configured queries*)
END_VAR
(*Structure Types*)
VAR
	HmiAudit : AuditHmiInterfaceType; (*HMI interface structure*)
	CustomEvent : ARRAY[0..MAX_CUSTOM_EVENTS] OF AuditCustomEventType; (*Custom events*)
	AuditQuery : {REDUND_UNREPLICABLE} AuditQueryType; (*Query results and status*)
	AuditTrailConfig : MpAuditTrailConfigType; (*Configuration structure for changing archiving setup*)
	MpAuditTrailUIConnect : MpAuditTrailUIConnectType; (*MpAuditUI connection to the HMI*)
END_VAR
(*Variables*)
VAR
	i : USINT; (*Index for loops*)
	ident : UDINT; (*Identifier for task deployment*)
	VariableMonitorExample : REAL; (*Used for the variable monitor example*)
END_VAR
VAR RETAIN
	ArchiveSettingsRetain : AuditArchiveParType; (*Store settings in retain memory to be applied after boot*)
END_VAR
```

#### HMIActions.st - Supporting code for the HMI interface
```iecst
ACTION ArchiveExport:

	// Assign variables to exchange with the HMI
	MpAuditTrailSys.ExportArchive := HmiAudit.Commands.ExportArchives;
	HmiAudit.Status.ArchiveAvailable := MpAuditTrailSys.ArchiveAvailable;
	HmiAudit.Status.NumberOfArchives := MpAuditTrailSys.Info.NumberArchives;

	IF (HmiAudit.Commands.ExportArchives AND MpAuditTrailSys.CommandDone) THEN
		HmiAudit.Commands.ExportArchives := FALSE;
	END_IF

END_ACTION

ACTION ArchiveSettings:

	// Audit Trail Config implementation
	IF (HmiAudit.Commands.SaveConfig) THEN
		HmiAudit.Commands.SaveConfig := FALSE;
		SaveAuditConfiguration;
		MpAuditTrailConfigSys.Save := TRUE;
	END_IF

	// After the configuration has been changed the AuditTrail is reset (disabled). This re-enables the component
	IF NOT MpAuditTrailSys.Active THEN
		MpAuditTrailSys.Enable := TRUE;
	END_IF

END_ACTION

ACTION SaveAuditConfiguration:

	// Assign current parameters from the HMI structure to AuditTrail configuration before saving it
	AuditTrailConfig.Archive.Time := UDINT_TO_TOD((((USINT_TO_UDINT(HmiAudit.Parameters.ArchiveSettings.Hour) * 60) +
	HmiAudit.Parameters.ArchiveSettings.Minute) * 60) * 1000);
	AuditTrailConfig.Archive.Enable := HmiAudit.Parameters.ArchiveSettings.Enable;
	AuditTrailConfig.Archive.MaxSize := HmiAudit.Parameters.ArchiveSettings.MaxSize;
	AuditTrailConfig.Archive.Mode := HmiAudit.Parameters.ArchiveSettings.Mode;
	AuditTrailConfig.Export.FileType := HmiAudit.Parameters.ArchiveSettings.FileType;

	// Save current archive setings to retain variable
	ArchiveSettingsRetain := HmiAudit.Parameters.ArchiveSettings;

 END_ACTION

ACTION LoadAuditConfiguration:

	// Assign current parameters from the configuration to the HMI structure
	HmiAudit.Parameters.ArchiveSettings.Hour := UDINT_TO_USINT(TOD_TO_UDINT(AuditTrailConfig.Archive.Time) / 1000 / 60 / 60);
	HmiAudit.Parameters.ArchiveSettings.Minute := UDINT_TO_USINT(TOD_TO_UDINT(AuditTrailConfig.Archive.Time) / 1000 / 60) -
													(HmiAudit.Parameters.ArchiveSettings.Hour * 60);
	HmiAudit.Parameters.ArchiveSettings.Enable := AuditTrailConfig.Archive.Enable;
	HmiAudit.Parameters.ArchiveSettings.MaxSize := AuditTrailConfig.Archive.MaxSize;
	HmiAudit.Parameters.ArchiveSettings.Mode := AuditTrailConfig.Archive.Mode;
	HmiAudit.Parameters.ArchiveSettings.FileType := AuditTrailConfig.Export.FileType;

END_ACTION

ACTION QueryTableConfig:

	// Configure visible list
	HmiAudit.Status.TableConfig[0] := '{ "specRows": [{"from":';
	HmiAudit.Status.Query.QueryCount := 0;
	FOR i := 0 TO 9 DO
		IF HmiAudit.Status.Query.Text[i] <> "" THEN
			HmiAudit.Status.Query.QueryCount := i + 1;
		END_IF
	END_FOR
	brsitoa((HmiAudit.Status.Query.QueryCount), ADR(HmiAudit.Status.TableConfig[0]) + brsstrlen(ADR(HmiAudit.Status.TableConfig[0])));
	brsstrcat(ADR(HmiAudit.Status.TableConfig[0]), ADR(',"to":19, "visible":false}]'));

	// Hide operator column for the recipe query
	IF (HmiAudit.Status.Query.Option = 0) THEN
		brsstrcat(ADR(HmiAudit.Status.TableConfig[0]), ADR(', "specColumns": [ {"from":2, "to":2, "visible":true}]'));
	ELSIF (HmiAudit.Status.Query.Option = 1) THEN
		brsstrcat(ADR(HmiAudit.Status.TableConfig[0]), ADR(', "specColumns": [ {"from":2, "to":2, "visible":false}]'));
	END_IF

	brsstrcat(ADR(HmiAudit.Status.TableConfig[0]), ADR('}'));

END_ACTION
```

#### ExecuteQuery.st - Runs a query
```iecst
ACTION ExecuteQuery:

	// Initialize mapp function block
	QueryUserEvents.MpLink := ADR(gMpLinkAuditTrail);
	QueryUserEvents.Enable := TRUE;
	QueryUserEvents.Name := ADR(HmiAudit.Status.Query.Name);
	QueryUserEvents.Language := ADR('en');
	QueryUserEvents();

	CASE (AuditQuery.State) OF
		ACTIVE_AUDIT_WAIT:
			// Wait until the RunQuery command is triggered from the HMI.
			// If you prefer that the query runs anytime new data is available, then uncomment line 15 and comment out line 16 and delete
			// the "Run query" button from the HMI.
			//IF (AuditQuery.LastUpdateCount <> AuditQuery.UpdateCount) THEN
			IF (HmiAudit.Commands.RunQuery) THEN
				// Call the custom event function when the query execution is triggered
				MpAuditCustomEvent(gMpLinkCustomEvents,CustomEvent[2].Type,CustomEvent[2].Msg,CustomEvent[2].Comment);
				brsmemset(ADR(AuditQuery.Audits[0]), 0, SIZEOF(AuditQuery.Audits));
				AuditQuery.LastUpdateCount := AuditQuery.UpdateCount;
				QueryUserEvents.Execute := TRUE;
				HmiAudit.Commands.RunQuery := FALSE;
				IF (HmiAudit.Status.Query.Name = 'UserEvents') THEN
					HmiAudit.Status.Query.Option := 0;
				ELSIF (HmiAudit.Status.Query.Name = 'RecipeEvents') THEN
					HmiAudit.Status.Query.Option := 1;
				END_IF

				AuditQuery.State := ACTIVE_AUDIT_QUERY;
			END_IF

		ACTIVE_AUDIT_QUERY:
			// If the number of query results is less than MAX_QUERY_RESULTS, return to the wait state
			IF ((QueryUserEvents.CommandDone) AND (NOT QueryUserEvents.Info.HasMoreRows)) THEN
				// Call the custom event function when the query execution is done
				MpAuditCustomEvent(gMpLinkCustomEvents,"Cmd Done","Executing the query command has finished","For additional information check the logger.");
				QueryUserEvents.Execute := FALSE;
				QueryUserEvents.Next := FALSE;
				AuditQuery.State := ACTIVE_AUDIT_WAIT;
				// If the number of query results is more than MAX_QUERY_RESULTS, then query the next set of results
			ELSIF ((QueryUserEvents.CommandDone) AND (QueryUserEvents.Info.HasMoreRows)) THEN
				QueryUserEvents.Next := FALSE;
				AuditQuery.State := ACTIVE_AUDIT_NEXT;
			END_IF

		ACTIVE_AUDIT_NEXT:
			IF (AuditQuery.Next) THEN
				// By default, AuditQuery.Alarms has 20 elements, so it can hold 20 query results at a time (MAX_QUERY_RESULTS = 19).
				// If AuditQuery.Next is true, this means the query result is more than 20 alarms.
				// If you want to save the data for the first 20 alarms, add code here to copy AuditQuery.Alarms to another location.
				// Otherwise, the older alarms in the query will get overwritten with the newest entries here.
				brsmemset(ADR(AuditQuery.Audits[0]), 0, SIZEOF(AuditQuery.Audits));
				AuditQuery.Next := FALSE;
				QueryUserEvents.Next := TRUE;
				AuditQuery.State := ACTIVE_AUDIT_QUERY;
			END_IF
	END_CASE

	// Convert the query results into arrays that can easily be bound to the Table widget in mapp View
	FOR i := 0 TO MAX_QUERY_RESULTS DO
		HmiAudit.Status.Query.EvTime[i] := AuditQuery.Audits[i].EvTime;
		HmiAudit.Status.Query.Op[i] := AuditQuery.Audits[i].Op;
		HmiAudit.Status.Query.Text[i] := AuditQuery.Audits[i].Text;
		HmiAudit.Status.Query.DText[i] := AuditQuery.Audits[i].DText;
	END_FOR

END_ACTION
```

#### ChangeConfiguration.st - Modifies the archive configuration at runtime
```iecst
ACTION ChangeConfiguration:

	MpAuditTrailConfigSys.MpLink := ADR(gMpLinkAuditTrail);
	MpAuditTrailConfigSys.Configuration := ADR(AuditTrailConfig);

	IF (MpAuditTrailConfigSys.Error = TRUE) THEN
		IF (MpAuditTrailConfigSys.StatusID = mpAUDIT_ERR_CONFIG_LOAD) THEN
			LoadAuditConfiguration;
		END_IF
		MpAuditTrailConfigSys.Load := FALSE;
		MpAuditTrailConfigSys.Save := FALSE;
		MpAuditTrailConfigSys.ErrorReset := TRUE;
	END_IF

	MpAuditTrailConfigSys();
	MpAuditTrailConfigSys.ErrorReset := FALSE;

	IF (MpAuditTrailConfigSys.CommandDone = TRUE) THEN
		IF (MpAuditTrailConfigSys.Load = TRUE) THEN
			LoadAuditConfiguration;
		END_IF
		// after save the AuditTrail needs to restart
		IF (MpAuditTrailConfigSys.Save = TRUE) THEN
			MpAuditTrailSys.Enable := FALSE;
		END_IF
		MpAuditTrailConfigSys.Load := FALSE;
		MpAuditTrailConfigSys.Save := FALSE;
	END_IF

END_ACTION
```

#### Variables.var - not listed in the package file held
```iecst
(*Function Blocks*)
VAR
	DirCreate_0 : DirCreate; (*DirCreate instance*)
END_VAR
(*Constants*)
VAR CONSTANT
	LOCAL_FOLDER : STRING[10] := 'Audit'; (*Folder name on the file device for UserX  files*)
END_VAR
(*Structure Types*)
(*Variables*)
```

#### Main.st - not listed in the package file held
```iecst
//***********************************************************************
// Copyright: B&R Industrial Automation GmbH
// Author: B&R Industrial Automation GmbH
// Created: Sept 1, 2022
// Description: Task for audit management.
//***********************************************************************

PROGRAM _INIT

	// Create folder for this component on the user file device
	DirCreate_0(enable := TRUE, pDevice := ADR('UserPartition'), pName := ADR(LOCAL_FOLDER));

	// Check if folder already exist and if so disabled the function block call
	IF DirCreate_0.status = fiERR_DIR_ALREADY_EXIST THEN
		DirCreate_0(enable := FALSE);
	END_IF

END_PROGRAM

PROGRAM _CYCLIC
	(* Insert code here *)

END_PROGRAM

PROGRAM _EXIT
	(* Insert code here *)

END_PROGRAM
```


### Package Logical/Infrastructure/Report - Package for mapp Report Framework

### Program Logical/Infrastructure/Report/ReportMgr (IEC) - Report Manager

#### ReportMgr.st - Init, cyclic, exit code
```iecst
//***********************************************************************
// Copyright: B&R Industrial Automation GmbH
// Author: B&R Industrial Automation GmbH
// Created: Dec 1, 2022
// Description: Task for generating reports.
//***********************************************************************

PROGRAM _INIT

	// Create folder for this component on the user file device
	DirCreateReport(enable := TRUE, pDevice := ADR('mappReportFiles'), pName := ADR('/'));

	// Wait for DirCreateReport to complete.
	WHILE (DirCreateReport.status = ERR_FUB_BUSY) DO
		DirCreateReport();
	END_WHILE

	// Check if folder already exist and if so disabled the function block call
	IF DirCreateReport.status = fiERR_DIR_ALREADY_EXIST OR (DirCreateReport.status = ERR_OK) THEN
		DirCreateReport(enable := FALSE);
	END_IF

	// Initialize mapp function blocks
	MpReportCoreSys.Language := ADR('en');
	MpReportCoreSys.DeviceName := ADR('mappReportFiles');
	MpReportCoreSys.MpLink := ADR(gMpLinkSimpleReport);
	MpReportCoreSys.Name := ADR(HmiReport.Parameters.Name);
	HmiReport.Parameters.Name := 'SimpleReport';
	HmiReport.Parameters.SortType := 'NameAsc';
	MpReportCoreSys();

	MpFileManagerUIConnect.DeviceList.DeviceNames[0] := 'mappReportFiles';
	MpFileManagerUIConnect.DeviceList.DeviceNames[1] := '';
	MpFileManagerUIConnect.DeviceList.DeviceNames[2] := '';
	MpFileManagerUIConnect.DeviceList.DeviceNames[3] := '';
	MpFileManagerUIConnect.DeviceList.DeviceNames[4] := '';
	MpFileManagerUIConnect.DeviceList.DeviceNames[5] := '';
	MpFileManagerUIConnect.DeviceList.DeviceNames[6] := '';
	MpFileManagerUIConnect.DeviceList.DeviceNames[7] := '';
	MpFileManagerUIConnect.DeviceList.DeviceNames[8] := '';
	MpFileManagerUIConnect.DeviceList.DeviceNames[9] := '';

	MpFileManagerUIReport.MpLink := ADR(gMpLinkFileManagerUIReport);
	MpFileManagerUIReport.UIConnect := ADR(MpFileManagerUIConnect);
	MpFileManagerUIReport.UISetup.FileListSize := SIZEOF(MpFileManagerUIConnect.File.List.Items) / SIZEOF(MpFileManagerUIConnect.File.List.Items[0]);
	MpFileManagerUIReport.Enable := TRUE;
	MpFileManagerUIReport();

	// Fill an array to create example data for the example report
	TimeIndex := 0;
	FOR i:=0 TO ((SIZEOF(ReportExample.SimpleReport.OeeLine[0].TemperatureSample.TimeStamp)/SIZEOF(ReportExample.SimpleReport.OeeLine[0].TemperatureSample.TimeStamp[0])) - 1) DO
		ReportExample.SimpleReport.OeeLine[0].TemperatureSample.TimeStamp[i] := TimeIndex;
		ReportExample.SimpleReport.OeeLine[1].TemperatureSample.TimeStamp[i] := TimeIndex;
		ReportExample.SimpleReport.OeeLine[2].TemperatureSample.TimeStamp[i] := TimeIndex;
		ReportExample.AdvancedReport.OeeLine[0].TemperatureSample.TimeStamp[i] := TimeIndex;
		ReportExample.AdvancedReport.OeeLine[1].TemperatureSample.TimeStamp[i] := TimeIndex;
		ReportExample.AdvancedReport.OeeLine[2].TemperatureSample.TimeStamp[i] := TimeIndex;
		TimeIndex := TimeIndex + 15;
	END_FOR

	// Ficticious number to serve as an example in the report
	ReportExample.AdvancedReport.BatchNumber := 325454685;

END_PROGRAM

PROGRAM _CYCLIC

	// Once a report has been generated, clear the generate command
	IF MpReportCoreSys.CommandDone THEN
		MpFileManagerUIConnect.File.Refresh := TRUE;
		HmiReport.Commands.Generate := FALSE;
	END_IF

	// Call all cyclic actions
	ReportFormat;
	ReportFileExplorer;

	// Generate command
	MpReportCoreSys.Generate := HmiReport.Commands.Generate;
	MpReportCoreSys.Name := ADR(HmiReport.Parameters.Name);

	// Assign address references
	MpFileManagerUIReport.UIConnect := ADR(MpFileManagerUIConnect);
	MpFileManagerUIReport.MpLink := ADR(gMpLinkFileManagerUIReport);
	MpFileManagerUIReport.UIConnect := ADR(MpFileManagerUIConnect);

	// Call function blocks
	MpReportCoreSys();
	MpFileManagerUIReport();

END_PROGRAM

PROGRAM _EXIT

	// Disable the function blocks to unlink the MpLinks
	MpReportCoreSys.Enable := FALSE;
	MpFileManagerUIReport.Enable := FALSE;

	// Call function blocks
	MpReportCoreSys();
	MpFileManagerUIReport();

END_PROGRAM
```
